C01838=1166.104,19.799,-47.480,-179.912,6.031,149.056
C01839=1166.100,20.048,-47.495,-179.910,6.031,149.055
C01840=1166.094,20.297,-47.509,-179.907,6.032,149.055
C01841=1166.089,20.547,-47.523,-179.905,6.033,149.054
C01842=1166.084,20.797,-47.538,-179.902,6.033,149.053
C01843=1166.078,21.047,-47.553,-179.899,6.034,149.053
C01844=1166.073,21.297,-47.567,-179.897,6.035,149.052
C01845=1166.069,21.546,-47.582,-179.894,6.036,149.052
C01846=1166.063,21.795,-47.596,-179.892,6.037,149.051
C01847=1166.058,22.044,-47.610,-179.889,6.037,149.051
C01848=1166.053,22.294,-47.624,-179.887,6.038,149.050
C01849=1166.048,22.544,-47.639,-179.884,6.039,149.049
C01850=1166.044,22.793,-47.654,-179.881,6.040,149.049
C01851=1166.038,23.043,-47.668,-179.879,6.041,149.048
C01852=1166.033,23.293,-47.683,-179.877,6.041,149.048
C01853=1166.028,23.542,-47.697,-179.874,6.042,149.047
C01854=1166.023,23.791,-47.712,-179.871,6.043,149.046
C01855=1166.018,24.040,-47.726,-179.869,6.044,149.046
C01856=1166.013,24.290,-47.740,-179.866,6.044,149.045
C01857=1166.008,24.540,-47.754,-179.864,6.045,149.045
C01858=1166.003,24.789,-47.770,-179.862,6.046,149.044
C01859=1165.998,25.039,-47.784,-179.858,6.047,149.043
C01860=1165.993,25.289,-47.799,-179.856,6.048,149.043
C01861=1165.988,25.538,-47.814,-179.853,6.048,149.042
C01862=1165.983,25.787,-47.828,-179.851,6.049,149.042
C01863=1165.977,26.037,-47.843,-179.849,6.050,149.041
C01864=1165.973,26.287,-47.858,-179.846,6.051,149.041
C01865=1165.968,26.536,-47.872,-179.843,6.052,149.040
C01866=1165.963,26.786,-47.886,-179.841,6.052,149.039
C01867=1165.957,27.035,-47.901,-179.838,6.053,149.039
C01868=1165.952,27.284,-47.916,-179.835,6.054,149.038
C01869=1165.947,27.534,-47.930,-179.833,6.055,149.038
C01870=1165.942,27.803,-47.946,-179.830,6.056,149.037
C01871=1165.936,28.072,-47.962,-179.827,6.057,149.036
C01872=1165.931,28.341,-47.978,-179.825,6.058,149.036
C01873=1165.925,28.610,-47.994,-179.822,6.058,149.035
C01874=1165.920,28.859,-48.009,-179.819,6.060,149.035
C01875=1165.915,29.109,-48.023,-179.817,6.060,149.034
C01876=1165.911,29.358,-48.038,-179.814,6.061,149.034
C01877=1165.905,29.608,-48.053,-179.812,6.062,149.033
C01878=1165.900,29.857,-48.068,-179.809,6.062,149.032
C01879=1165.895,30.107,-48.082,-179.807,6.064,149.032
C01880=1165.890,30.357,-48.097,-179.804,6.064,149.031
C01881=1165.885,30.606,-48.112,-179.801,6.065,149.031
C01882=1165.880,30.855,-48.127,-179.799,6.066,149.030
C01883=1165.875,31.105,-48.142,-179.796,6.067,149.029
C01884=1165.870,31.354,-48.157,-179.794,6.068,149.029
C01885=1165.865,31.604,-48.171,-179.791,6.068,149.028
C01886=1165.860,31.853,-48.187,-179.789,6.069,149.028
C01887=1165.855,32.103,-48.201,-179.786,6.070,149.027
C01888=1165.850,32.352,-48.216,-179.784,6.071,149.027
C01889=1165.844,32.602,-48.231,-179.781,6.072,149.026
C01890=1165.840,32.851,-48.246,-179.779,6.073,149.026
C01891=1165.834,33.101,-48.261,-179.776,6.074,149.025
C01892=1165.829,33.350,-48.276,-179.773,6.074,149.024
C01893=1165.825,33.599,-48.291,-179.771,6.075,149.024
C01894=1165.820,33.850,-48.306,-179.768,6.076,149.023
C01895=1165.815,34.099,-48.321,-179.765,6.077,149.023
C01896=1165.810,34.348,-48.337,-179.763,6.078,149.022
C01897=1165.805,34.598,-48.351,-179.761,6.079,149.022
C01898=1165.799,34.847,-48.367,-179.758,6.079,149.021
C01899=1165.794,35.097,-48.381,-179.755,6.081,149.020
C01900=1165.790,35.346,-48.396,-179.753,6.081,149.020
C01901=1165.784,35.596,-48.412,-179.750,6.082,149.019
C01902=1165.780,35.845,-48.427,-179.747,6.084,149.019
C01903=1165.774,36.095,-48.441,-179.745,6.084,149.018
C01904=1165.769,36.344,-48.456,-179.742,6.085,149.018
C01905=1165.764,36.593,-48.472,-179.740,6.085,149.017
C01906=1165.760,36.844,-48.487,-179.737,6.087,149.016
C01907=1165.754,37.093,-48.502,-179.734,6.087,149.016
C01908=1165.750,37.342,-48.517,-179.732,6.088,149.015
C01909=1165.744,37.592,-48.533,-179.730,6.089,149.015
C01910=1165.739,37.841,-48.547,-179.727,6.090,149.014
C01911=1165.734,38.091,-48.563,-179.724,6.091,149.014
C01912=1165.729,38.340,-48.578,-179.722,6.092,149.013
C01913=1165.724,38.589,-48.593,-179.719,6.093,149.012
C01914=1165.719,38.840,-48.608,-179.717,6.094,149.012
C01915=1165.714,39.089,-48.623,-179.714,6.094,149.011
C01916=1165.709,39.338,-48.639,-179.711,6.096,149.011
C01917=1165.704,39.587,-48.654,-179.709,6.097,149.010
C01918=1165.699,39.837,-48.670,-179.706,6.097,149.010
C01919=1165.694,40.086,-48.685,-179.704,6.098,149.009
C01920=1165.688,40.336,-48.700,-179.701,6.100,149.009
C01921=1165.684,40.586,-48.715,-179.698,6.100,149.008
C01922=1165.679,40.835,-48.730,-179.696,6.101,149.007
C01923=1165.673,41.085,-48.746,-179.693,6.102,149.007
C01924=1165.669,41.334,-48.761,-179.690,6.103,149.006
C01925=1165.663,41.583,-48.777,-179.688,6.104,149.006
C01926=1165.659,41.833,-48.792,-179.685,6.105,149.005
C01927=1165.654,42.082,-48.808,-179.683,6.106,149.005
C01928=1165.649,42.332,-48.823,-179.680,6.106,149.004
C01929=1165.644,42.581,-48.837,-179.678,6.107,149.003
C01930=1165.638,42.831,-48.853,-179.675,6.108,149.003
C01931=1165.633,43.081,-48.869,-179.673,6.109,149.002
C01932=1165.629,43.330,-48.884,-179.670,6.110,149.002
C01933=1165.623,43.579,-48.900,-179.667,6.111,149.001
C01934=1165.618,43.829,-48.915,-179.665,6.112,149.001
C01935=1165.613,44.078,-48.930,-179.662,6.113,149.000
C01936=1165.609,44.328,-48.946,-179.659,6.114,148.999
C01937=1165.603,44.577,-48.962,-179.657,6.115,148.999
C01938=1165.599,44.827,-48.977,-179.654,6.115,148.998
C01939=1165.593,45.076,-48.992,-179.652,6.117,148.998
C01940=1165.588,45.326,-49.008,-179.649,6.118,148.997
C01941=1165.584,45.575,-49.023,-179.647,6.118,148.997
C01942=1165.578,45.825,-49.039,-179.644,6.120,148.996
C01943=1165.573,46.074,-49.054,-179.641,6.121,148.996
C01944=1165.568,46.323,-49.071,-179.639,6.121,148.995
C01945=1165.564,46.572,-49.086,-179.636,6.123,148.995
C01946=1165.558,46.822,-49.102,-179.633,6.123,148.994
C01947=1165.554,47.072,-49.118,-179.631,6.124,148.993
C01948=1165.548,47.321,-49.133,-179.628,6.125,148.993
C01949=1165.544,47.570,-49.148,-179.626,6.126,148.992
C01950=1165.538,47.820,-49.164,-179.623,6.127,148.992
C01951=1165.533,48.070,-49.180,-179.621,6.128,148.991
C01952=1165.528,48.319,-49.195,-179.618,6.129,148.991
C01953=1165.524,48.568,-49.211,-179.616,6.130,148.990
C01954=1165.519,48.818,-49.227,-179.613,6.131,148.989
C01955=1165.514,49.067,-49.243,-179.610,6.132,148.989
C01956=1165.508,49.317,-49.258,-179.608,6.132,148.988
C01957=1165.503,49.567,-49.274,-179.605,6.134,148.988
C01958=1165.499,49.816,-49.289,-179.602,6.135,148.987
C01959=1165.494,50.065,-49.305,-179.600,6.136,148.987
C01960=1165.489,50.315,-49.321,-179.597,6.137,148.986
C01961=1165.483,50.564,-49.337,-179.595,6.138,148.986
C01962=1165.478,50.814,-49.353,-179.592,6.139,148.985
C01963=1165.474,51.063,-49.369,-179.589,6.140,148.985
C01964=1165.469,51.312,-49.384,-179.587,6.140,148.984
C01965=1165.464,51.562,-49.400,-179.584,6.142,148.983
C01966=1165.459,51.812,-49.416,-179.581,6.142,148.983
C01967=1165.454,52.061,-49.432,-179.579,6.143,148.982
C01968=1165.449,52.311,-49.448,-179.576,6.145,148.982
C01969=1165.444,52.560,-49.464,-179.574,6.145,148.981
C01970=1165.438,52.809,-49.480,-179.571,6.147,148.981
C01971=1165.434,53.059,-49.496,-179.568,6.148,148.980
C01972=1165.428,53.308,-49.511,-179.566,6.148,148.979
C01973=1165.424,53.557,-49.527,-179.563,6.150,148.979
C01974=1165.419,53.826,-49.545,-179.560,6.150,148.978
C01975=1165.413,54.094,-49.562,-179.557,6.152,148.978
C01976=1165.408,54.363,-49.579,-179.555,6.152,148.977
C01977=1165.402,54.631,-49.596,-179.552,6.154,148.977
C01978=1165.398,54.882,-49.612,-179.549,6.154,148.976
C01979=1165.392,55.130,-49.628,-179.546,6.156,148.975
C01980=1165.388,55.380,-49.644,-179.544,6.156,148.975
C01981=1165.383,55.629,-49.660,-179.541,6.158,148.974
C01982=1165.378,55.879,-49.676,-179.539,6.159,148.974
C01983=1165.373,56.128,-49.692,-179.536,6.159,148.973
C01984=1165.367,56.377,-49.708,-179.534,6.161,148.973
C01985=1165.363,56.628,-49.724,-179.531,6.162,148.972
C01986=1165.357,56.876,-49.740,-179.528,6.163,148.972
C01987=1165.353,57.126,-49.756,-179.526,6.164,148.971
C01988=1165.348,57.375,-49.772,-179.523,6.165,148.971
C01989=1165.343,57.625,-49.788,-179.520,6.166,148.970
C01990=1165.338,57.874,-49.805,-179.518,6.167,148.969
C01991=1165.333,58.124,-49.821,-179.515,6.168,148.969
C01992=1165.328,58.373,-49.837,-179.513,6.169,148.968
C01993=1165.322,58.623,-49.854,-179.510,6.170,148.968
C01994=1165.317,58.872,-49.870,-179.507,6.171,148.967
C01995=1165.312,59.122,-49.886,-179.505,6.172,148.967
C01996=1165.307,59.371,-49.902,-179.502,6.173,148.966
C01997=1165.303,59.621,-49.919,-179.499,6.174,148.966
C01998=1165.298,59.870,-49.934,-179.497,6.176,148.965
C01999=1165.293,60.119,-49.951,-179.494,6.176,148.964
C02000=1165.288,60.369,-49.967,-179.492,6.177,148.964
C02001=1165.283,60.618,-49.983,-179.489,6.179,148.964
C02002=1165.278,60.867,-50.000,-179.486,6.179,148.963
C02003=1165.273,61.117,-50.016,-179.484,6.181,148.962
C02004=1165.268,61.366,-50.032,-179.481,6.181,148.962
C02005=1165.263,61.616,-50.048,-179.478,6.183,148.961
C02006=1165.258,61.865,-50.065,-179.476,6.183,148.961
C02007=1165.253,62.115,-50.081,-179.473,6.184,148.960
C02008=1165.248,62.364,-50.097,-179.470,6.186,148.960
C02009=1165.243,62.614,-50.114,-179.468,6.187,148.959
C02010=1165.238,62.862,-50.130,-179.465,6.188,148.958
C02011=1165.233,63.112,-50.147,-179.463,6.189,148.958
C02012=1165.228,63.362,-50.163,-179.460,6.190,148.958
C02013=1165.223,63.611,-50.179,-179.457,6.191,148.957
C02014=1165.219,63.861,-50.196,-179.455,6.193,148.957
C02015=1165.213,64.110,-50.212,-179.452,6.193,148.956
C02016=1165.209,64.359,-50.228,-179.450,6.194,148.955
C02017=1165.203,64.609,-50.245,-179.447,6.195,148.955
C02018=1165.198,64.858,-50.262,-179.444,6.196,148.954
C02019=1165.194,65.108,-50.278,-179.441,6.197,148.954
C02020=1165.189,65.357,-50.294,-179.439,6.198,148.953
C02021=1165.183,65.607,-50.311,-179.436,6.200,148.953
C02022=1165.178,65.855,-50.328,-179.434,6.200,148.952
C02023=1165.174,66.105,-50.344,-179.431,6.202,148.952
C02024=1165.169,66.354,-50.361,-179.428,6.203,148.951
C02025=1165.163,66.604,-50.377,-179.426,6.204,148.951
C02026=1165.159,66.854,-50.394,-179.423,6.205,148.950
C02027=1165.154,67.103,-50.411,-179.420,6.207,148.950
C02028=1165.149,67.352,-50.427,-179.418,6.207,148.949
C02029=1165.144,67.602,-50.444,-179.415,6.209,148.948
C02030=1165.139,67.850,-50.460,-179.412,6.209,148.948
C02031=1165.134,68.100,-50.477,-179.410,6.210,148.947
C02032=1165.130,68.350,-50.493,-179.407,6.212,148.947
C02033=1165.124,68.599,-50.510,-179.405,6.212,148.946
C02034=1165.119,68.849,-50.527,-179.402,6.214,148.946
C02035=1165.115,69.098,-50.543,-179.399,6.215,148.945
C02036=1165.109,69.347,-50.560,-179.397,6.216,148.945
C02037=1165.105,69.597,-50.577,-179.394,6.217,148.944
C02038=1165.100,69.846,-50.594,-179.391,6.218,148.944
C02039=1165.094,70.095,-50.610,-179.389,6.219,148.943
C02040=1165.090,70.345,-50.627,-179.386,6.221,148.943
C02041=1165.085,70.595,-50.644,-179.384,6.221,148.942
C02042=1165.080,70.844,-50.661,-179.381,6.223,148.941
C02043=1165.075,71.093,-50.677,-179.378,6.224,148.941
C02044=1165.070,71.343,-50.695,-179.375,6.225,148.940
C02045=1165.065,71.592,-50.711,-179.373,6.226,148.940
C02046=1165.060,71.841,-50.728,-179.370,6.228,148.939
C02047=1165.055,72.091,-50.745,-179.368,6.228,148.939
C02048=1165.050,72.340,-50.762,-179.365,6.230,148.938
C02049=1165.045,72.589,-50.778,-179.362,6.230,148.938
C02050=1165.040,72.839,-50.795,-179.360,6.232,148.937
C02051=1165.035,73.089,-50.812,-179.357,6.232,148.937
C02052=1165.031,73.337,-50.830,-179.354,6.234,148.936
C02053=1165.026,73.586,-50.846,-179.352,6.235,148.936
C02054=1165.021,73.836,-50.863,-179.349,6.236,148.935
C02055=1165.016,74.085,-50.880,-179.347,6.237,148.935
C02056=1165.011,74.335,-50.897,-179.343,6.239,148.934
C02057=1165.006,74.584,-50.914,-179.341,6.239,148.934
C02058=1165.001,74.834,-50.931,-179.339,6.241,148.933
C02059=1164.996,75.083,-50.947,-179.336,6.242,148.933
C02060=1164.991,75.333,-50.965,-179.333,6.243,148.932
C02061=1164.987,75.582,-50.982,-179.330,6.245,148.931
C02062=1164.981,75.831,-50.999,-179.328,6.246,148.931
C02063=1164.976,76.081,-51.016,-179.325,6.247,148.931
C02064=1164.971,76.330,-51.033,-179.322,6.248,148.930
C02065=1164.967,76.579,-51.050,-179.320,6.249,148.930
C02066=1164.962,76.829,-51.068,-179.317,6.250,148.929
C02067=1164.957,77.078,-51.084,-179.314,6.252,148.928
C02068=1164.951,77.328,-51.101,-179.312,6.252,148.928
C02069=1164.947,77.577,-51.119,-179.309,6.254,148.927
C02070=1164.942,77.826,-51.136,-179.307,6.255,148.927
C02071=1164.937,78.076,-51.153,-179.304,6.256,148.926
C02072=1164.932,78.324,-51.170,-179.302,6.257,148.926
C02073=1164.927,78.574,-51.187,-179.299,6.259,148.925
C02074=1164.922,78.823,-51.204,-179.296,6.260,148.925
C02075=1164.917,79.073,-51.221,-179.293,6.261,148.924
C02076=1164.912,79.322,-51.239,-179.290,6.262,148.924
C02077=1164.908,79.572,-51.256,-179.288,6.263,148.923
C02078=1164.902,79.840,-51.274,-179.285,6.264,148.923
C02079=1164.897,80.108,-51.294,-179.282,6.266,148.922
C02080=1164.892,80.377,-51.312,-179.280,6.267,148.922
C02081=1164.886,80.645,-51.330,-179.277,6.268,148.921
C02082=1164.881,80.895,-51.347,-179.274,6.270,148.920
C02083=1164.877,81.144,-51.365,-179.271,6.270,148.920
C02084=1164.871,81.394,-51.382,-179.269,6.272,148.920
C02085=1164.867,81.643,-51.400,-179.266,6.273,148.919
C02086=1164.862,81.892,-51.417,-179.263,6.274,148.919
C02087=1164.857,82.141,-51.435,-179.260,6.276,148.918
C02088=1164.851,82.390,-51.452,-179.258,6.277,148.917
C02089=1164.847,82.640,-51.468,-179.255,6.278,148.917
C02090=1164.842,82.889,-51.486,-179.253,6.279,148.916
C02091=1164.837,83.139,-51.503,-179.250,6.280,148.916
C02092=1164.832,83.388,-51.521,-179.247,6.281,148.915
C02093=1164.827,83.638,-51.538,-179.245,6.283,148.915
C02094=1164.822,83.887,-51.556,-179.242,6.284,148.914
C02095=1164.817,84.137,-51.573,-179.239,6.285,148.914
C02096=1164.812,84.386,-51.591,-179.236,6.287,148.913
C02097=1164.808,84.635,-51.609,-179.234,6.287,148.913
C02098=1164.803,84.884,-51.626,-179.231,6.289,148.912
C02099=1164.798,85.134,-51.644,-179.228,6.290,148.912
C02100=1164.793,85.383,-51.661,-179.226,6.291,148.911
C02101=1164.789,85.632,-51.679,-179.223,6.293,148.911
C02102=1164.783,85.882,-51.696,-179.221,6.294,148.910
C02103=1164.778,86.131,-51.714,-179.218,6.295,148.910
C02104=1164.773,86.380,-51.731,-179.215,6.297,148.909
C02105=1164.768,86.629,-51.749,-179.213,6.298,148.909
C02106=1164.764,86.878,-51.766,-179.210,6.299,148.908
C02107=1164.758,87.128,-51.783,-179.207,6.300,148.908
C02108=1164.753,87.377,-51.801,-179.205,6.301,148.907
C02109=1164.748,87.626,-51.819,-179.201,6.303,148.907
C02110=1164.743,87.876,-51.837,-179.199,6.304,148.906
C02111=1164.738,88.125,-51.855,-179.197,6.305,148.906
C02112=1164.734,88.374,-51.872,-179.194,6.306,148.905
C02113=1164.729,88.624,-51.890,-179.191,6.308,148.905
C02114=1164.724,88.873,-51.907,-179.188,6.309,148.904
C02115=1164.719,89.122,-51.925,-179.186,6.310,148.904
C02116=1164.714,89.372,-51.943,-179.183,6.311,148.903
C02117=1164.710,89.622,-51.961,-179.180,6.313,148.903
C02118=1164.705,89.871,-51.979,-179.178,6.314,148.902
C02119=1164.700,90.121,-51.997,-179.175,6.315,148.902
C02120=1164.696,90.369,-52.014,-179.173,6.316,148.901
C02121=1164.691,90.619,-52.032,-179.170,6.318,148.901
C02122=1164.685,90.868,-52.049,-179.167,6.319,148.900
C02123=1164.681,91.118,-52.067,-179.164,6.320,148.900
C02124=1164.676,91.367,-52.085,-179.162,6.322,148.899
C02125=1164.671,91.616,-52.103,-179.159,6.323,148.899
C02126=1164.666,91.865,-52.121,-179.156,6.324,148.898
C02127=1164.661,92.115,-52.139,-179.154,6.325,148.898
C02128=1164.656,92.364,-52.157,-179.151,6.326,148.897
C02129=1164.651,92.613,-52.175,-179.148,6.328,148.897
C02130=1164.646,92.862,-52.193,-179.146,6.329,148.896
C02131=1164.641,93.112,-52.211,-179.143,6.330,148.896
C02132=1164.637,93.361,-52.229,-179.140,6.332,148.895
C02133=1164.632,93.611,-52.247,-179.137,6.333,148.895
C02134=1164.627,93.860,-52.265,-179.135,6.334,148.894
C02135=1164.622,94.109,-52.283,-179.132,6.336,148.894
C02136=1164.617,94.359,-52.300,-179.129,6.337,148.893
C02137=1164.612,94.608,-52.318,-179.127,6.338,148.893
C02138=1164.607,94.857,-52.336,-179.124,6.340,148.892
C02139=1164.602,95.106,-52.354,-179.121,6.341,148.892
C02140=1164.597,95.355,-52.372,-179.119,6.342,148.891
C02141=1164.593,95.605,-52.390,-179.116,6.343,148.891
C02142=1164.588,95.855,-52.408,-179.113,6.345,148.890
C02143=1164.583,96.104,-52.426,-179.111,6.346,148.890
C02144=1164.578,96.353,-52.444,-179.108,6.348,148.890
C02145=1164.573,96.602,-52.462,-179.105,6.349,148.889
C02146=1164.567,96.852,-52.481,-179.103,6.350,148.889
C02147=1164.563,97.101,-52.499,-179.100,6.352,148.888
C02148=1164.558,97.351,-52.517,-179.097,6.353,148.887
C02149=1164.553,97.600,-52.535,-179.095,6.354,148.887
C02150=1164.549,97.848,-52.554,-179.092,6.356,148.887
C02151=1164.544,98.097,-52.572,-179.089,6.357,148.886
C02152=1164.539,98.347,-52.590,-179.087,6.358,148.886
C02153=1164.535,98.597,-52.608,-179.084,6.360,148.885
C02154=1164.530,98.846,-52.626,-179.081,6.361,148.885
C02155=1164.524,99.095,-52.645,-179.079,6.362,148.884
C02156=1164.519,99.344,-52.663,-179.076,6.363,148.884
C02157=1164.514,99.594,-52.681,-179.073,6.365,148.883
C02158=1164.510,99.843,-52.700,-179.071,6.366,148.883
C02159=1164.505,100.092,-52.718,-179.068,6.367,148.882
C02160=1164.500,100.341,-52.736,-179.065,6.369,148.882
C02161=1164.495,100.591,-52.754,-179.062,6.370,148.881
C02162=1164.490,100.841,-52.773,-179.060,6.371,148.881
C02163=1164.485,101.090,-52.791,-179.057,6.373,148.880
C02164=1164.481,101.338,-52.809,-179.055,6.375,148.880
C02165=1164.475,101.588,-52.828,-179.052,6.375,148.879
C02166=1164.470,101.837,-52.846,-179.049,6.377,148.879
C02167=1164.466,102.087,-52.864,-179.047,6.379,148.878
C02168=1164.461,102.335,-52.883,-179.044,6.379,148.878
C02169=1164.456,102.585,-52.901,-179.041,6.381,148.877
C02170=1164.451,102.835,-52.920,-179.038,6.383,148.877
C02171=1164.447,103.084,-52.938,-179.036,6.384,148.877
C02172=1164.442,103.332,-52.956,-179.033,6.385,148.876
C02173=1164.436,103.582,-52.975,-179.030,6.387,148.876
C02174=1164.432,103.832,-52.993,-179.028,6.388,148.875
C02175=1164.427,104.080,-53.012,-179.025,6.389,148.874
C02176=1164.422,104.330,-53.030,-179.022,6.391,148.874
C02177=1164.417,104.580,-53.049,-179.020,6.392,148.874
C02178=1164.413,104.828,-53.068,-179.017,6.394,148.873
C02179=1164.408,105.077,-53.086,-179.014,6.395,148.873
C02180=1164.403,105.326,-53.105,-179.012,6.396,148.872
C02181=1164.398,105.576,-53.123,-179.009,6.398,148.872
C02182=1164.392,105.845,-53.143,-179.006,6.399,148.871
C02183=1164.388,106.112,-53.163,-179.003,6.401,148.871
C02184=1164.382,106.382,-53.184,-179.000,6.402,148.870
C02185=1164.377,106.650,-53.203,-178.997,6.404,148.870
C02186=1164.372,106.899,-53.223,-178.995,6.405,148.869
C02187=1164.368,107.149,-53.241,-178.992,6.407,148.869
C02188=1164.363,107.397,-53.260,-178.989,6.408,148.868
C02189=1164.357,107.647,-53.278,-178.986,6.410,148.868
C02190=1164.353,107.896,-53.297,-178.984,6.411,148.867
C02191=1164.348,108.145,-53.316,-178.981,6.412,148.867
C02192=1164.343,108.394,-53.334,-178.978,6.414,148.866
C02193=1164.339,108.644,-53.353,-178.975,6.415,148.866
C02194=1164.333,108.893,-53.372,-178.973,6.416,148.866
C02195=1164.329,109.142,-53.390,-178.970,6.418,148.865
C02196=1164.324,109.391,-53.410,-178.967,6.419,148.865
C02197=1164.319,109.641,-53.428,-178.965,6.421,148.864
C02198=1164.314,109.890,-53.447,-178.963,6.422,148.864
C02199=1164.309,110.139,-53.465,-178.960,6.424,148.863
C02200=1164.304,110.388,-53.485,-178.957,6.425,148.863
C02201=1164.300,110.638,-53.504,-178.954,6.427,148.862
C02202=1164.295,110.887,-53.522,-178.952,6.428,148.862
C02203=1164.290,111.136,-53.541,-178.949,6.429,148.861
C02204=1164.285,111.385,-53.559,-178.946,6.431,148.861
C02205=1164.281,111.635,-53.579,-178.943,6.432,148.860
C02206=1164.275,111.884,-53.598,-178.940,6.434,148.860
C02207=1164.270,112.133,-53.616,-178.938,6.435,148.860
C02208=1164.266,112.383,-53.636,-178.935,6.436,148.859
C02209=1164.261,112.631,-53.655,-178.932,6.438,148.859
C02210=1164.256,112.881,-53.674,-178.930,6.440,148.858
C02211=1164.251,113.130,-53.692,-178.928,6.441,148.858
C02212=1164.247,113.380,-53.712,-178.924,6.442,148.857
C02213=1164.242,113.628,-53.731,-178.922,6.444,148.857
C02214=1164.237,113.878,-53.750,-178.919,6.446,148.856
C02215=1164.232,114.127,-53.769,-178.916,6.447,148.856
C02216=1164.228,114.376,-53.788,-178.914,6.448,148.855
C02217=1164.222,114.625,-53.807,-178.911,6.450,148.855
C02218=1164.218,114.875,-53.826,-178.908,6.451,148.854
C02219=1164.213,115.124,-53.845,-178.905,6.453,148.854
C02220=1164.208,115.374,-53.864,-178.903,6.455,148.854
C02221=1164.203,115.622,-53.883,-178.901,6.456,148.853
C02222=1164.199,115.872,-53.903,-178.897,6.457,148.853
C02223=1164.193,116.121,-53.922,-178.895,6.459,148.852
C02224=1164.189,116.370,-53.940,-178.892,6.460,148.852
C02225=1164.184,116.619,-53.960,-178.889,6.462,148.851
C02226=1164.179,116.869,-53.979,-178.887,6.463,148.851
C02227=1164.174,117.117,-53.998,-178.884,6.464,148.850
C02228=1164.169,117.367,-54.018,-178.881,6.466,148.850
C02229=1164.164,117.616,-54.037,-178.879,6.468,148.850
C02230=1164.160,117.865,-54.056,-178.876,6.470,148.849
C02231=1164.155,118.114,-54.075,-178.873,6.471,148.849
C02232=1164.150,118.364,-54.094,-178.870,6.472,148.848
C02233=1164.145,118.613,-54.113,-178.868,6.473,148.848
C02234=1164.140,118.862,-54.133,-178.865,6.475,148.847
C02235=1164.136,119.112,-54.152,-178.862,6.477,148.847
C02236=1164.130,119.361,-54.172,-178.860,6.479,148.847
C02237=1164.126,119.610,-54.191,-178.857,6.479,148.846
C02238=1164.121,119.859,-54.210,-178.854,6.481,148.845
C02239=1164.116,120.108,-54.230,-178.852,6.483,148.845
C02240=1164.111,120.358,-54.249,-178.849,6.484,148.845
C02241=1164.107,120.607,-54.268,-178.846,6.486,148.844
C02242=1164.102,120.856,-54.288,-178.843,6.487,148.844
C02243=1164.097,121.105,-54.307,-178.840,6.489,148.843
C02244=1164.092,121.355,-54.327,-178.838,6.490,148.843
C02245=1164.088,121.603,-54.346,-178.835,6.492,148.842
C02246=1164.083,121.852,-54.366,-178.833,6.494,148.842
C02247=1164.078,122.102,-54.385,-178.830,6.495,148.842
C02248=1164.073,122.350,-54.405,-178.827,6.497,148.841
C02249=1164.068,122.600,-54.424,-178.824,6.498,148.841
C02250=1164.063,122.850,-54.444,-178.822,6.499,148.840
C02251=1164.059,123.098,-54.463,-178.819,6.501,148.840
C02252=1164.054,123.348,-54.482,-178.817,6.503,148.839
C02253=1164.049,123.597,-54.502,-178.814,6.504,148.839
C02254=1164.044,123.846,-54.522,-178.811,6.506,148.838
C02255=1164.039,124.095,-54.542,-178.808,6.507,148.838
C02256=1164.035,124.345,-54.561,-178.805,6.509,148.838
C02257=1164.029,124.594,-54.581,-178.803,6.510,148.837
C02258=1164.025,124.843,-54.600,-178.800,6.512,148.837
C02259=1164.021,125.092,-54.620,-178.798,6.514,148.836
C02260=1164.016,125.341,-54.639,-178.794,6.515,148.836
C02261=1164.011,125.590,-54.659,-178.792,6.517,148.835
C02262=1164.006,125.840,-54.679,-178.789,6.518,148.835
C02263=1164.002,126.089,-54.699,-178.786,6.520,148.835
C02264=1163.996,126.338,-54.718,-178.784,6.522,148.834
C02265=1163.992,126.587,-54.738,-178.781,6.523,148.834
C02266=1163.987,126.837,-54.758,-178.779,6.524,148.833
C02267=1163.982,127.085,-54.778,-178.776,6.526,148.833
C02268=1163.977,127.335,-54.797,-178.773,6.528,148.832
C02269=1163.972,127.584,-54.817,-178.770,6.529,148.832
C02270=1163.968,127.833,-54.837,-178.767,6.531,148.832
C02271=1163.963,128.082,-54.857,-178.765,6.533,148.831
C02272=1163.958,128.331,-54.876,-178.762,6.534,148.831
C02273=1163.953,128.580,-54.897,-178.759,6.536,148.830
C02274=1163.949,128.830,-54.916,-178.757,6.537,148.830
C02275=1163.944,129.078,-54.936,-178.754,6.538,148.829
C02276=1163.939,129.328,-54.956,-178.751,6.540,148.829
C02277=1163.934,129.577,-54.976,-178.749,6.542,148.829
C02278=1163.930,129.826,-54.996,-178.746,6.544,148.828
C02279=1163.925,130.076,-55.016,-178.743,6.545,148.828
C02280=1163.920,130.324,-55.036,-178.740,6.547,148.827
C02281=1163.915,130.574,-55.055,-178.738,6.549,148.827
C02282=1163.911,130.823,-55.076,-178.735,6.550,148.826
C02283=1163.906,131.072,-55.095,-178.732,6.552,148.826
C02284=1163.901,131.320,-55.115,-178.729,6.554,148.826
C02285=1163.896,131.570,-55.135,-178.727,6.555,148.825
C02286=1163.891,131.839,-55.157,-178.724,6.557,148.825
C02287=1163.886,132.107,-55.178,-178.721,6.559,148.824
C02288=1163.880,132.376,-55.200,-178.718,6.560,148.824
C02289=1163.875,132.645,-55.221,-178.715,6.562,148.823
C02290=1163.871,132.894,-55.242,-178.712,6.564,148.823
C02291=1163.866,133.143,-55.262,-178.710,6.565,148.823
C02292=1163.861,133.392,-55.282,-178.707,6.567,148.822
C02293=1163.857,133.641,-55.303,-178.704,6.569,148.822
C02294=1163.851,133.890,-55.322,-178.701,6.570,148.821
C02295=1163.847,134.139,-55.342,-178.698,6.572,148.821
C02296=1163.842,134.389,-55.362,-178.696,6.574,148.820
C02297=1163.838,134.638,-55.382,-178.694,6.575,148.820
C02298=1163.832,134.887,-55.403,-178.691,6.576,148.820
C02299=1163.828,135.137,-55.423,-178.688,6.578,148.819
C02300=1163.823,135.385,-55.443,-178.685,6.580,148.819
C02301=1163.819,135.634,-55.464,-178.683,6.581,148.818
C02302=1163.813,135.883,-55.483,-178.680,6.583,148.818
C02303=1163.808,136.133,-55.504,-178.677,6.585,148.818
C02304=1163.804,136.382,-55.524,-178.675,6.587,148.817
C02305=1163.799,136.630,-55.545,-178.671,6.588,148.817
C02306=1163.795,136.880,-55.564,-178.669,6.590,148.816
C02307=1163.789,137.129,-55.585,-178.666,6.591,148.816
C02308=1163.785,137.378,-55.606,-178.663,6.593,148.816
C02309=1163.781,137.627,-55.626,-178.661,6.595,148.815
C02310=1163.776,137.877,-55.646,-178.658,6.597,148.815
C02311=1163.771,138.126,-55.667,-178.655,6.598,148.814
C02312=1163.766,138.375,-55.687,-178.653,6.600,148.814
C02313=1163.761,138.623,-55.707,-178.650,6.602,148.814
C02314=1163.756,138.872,-55.728,-178.647,6.604,148.813
C02315=1163.751,139.122,-55.748,-178.644,6.605,148.813
C02316=1163.747,139.371,-55.768,-178.642,6.607,148.812
C02317=1163.742,139.620,-55.789,-178.639,6.609,148.812
C02318=1163.737,139.869,-55.809,-178.636,6.611,148.812
C02319=1163.733,140.118,-55.830,-178.633,6.612,148.811
C02320=1163.728,140.367,-55.851,-178.630,6.614,148.811
C02321=1163.723,140.616,-55.871,-178.628,6.615,148.810
C02322=1163.718,140.866,-55.891,-178.625,6.617,148.810
C02323=1163.713,141.115,-55.912,-178.623,6.618,148.809
C02324=1163.709,141.364,-55.932,-178.620,6.620,148.809
C02325=1163.704,141.613,-55.952,-178.617,6.622,148.809
C02326=1163.699,141.862,-55.973,-178.615,6.623,148.808
C02327=1163.695,142.111,-55.994,-178.612,6.625,148.808
C02328=1163.690,142.361,-56.015,-178.609,6.627,148.808
C02329=1163.685,142.609,-56.035,-178.607,6.628,148.807
C02330=1163.680,142.859,-56.056,-178.604,6.630,148.807
C02331=1163.676,143.108,-56.076,-178.601,6.632,148.806
C02332=1163.671,143.357,-56.097,-178.599,6.634,148.806
C02333=1163.666,143.606,-56.118,-178.596,6.635,148.806
C02334=1163.662,143.855,-56.138,-178.593,6.637,148.805
C02335=1163.657,144.105,-56.159,-178.590,6.639,148.805
C02336=1163.653,144.354,-56.180,-178.588,6.641,148.804
C02337=1163.647,144.603,-56.201,-178.585,6.642,148.804
C02338=1163.643,144.852,-56.221,-178.582,6.644,148.804
C02339=1163.638,145.101,-56.243,-178.580,6.646,148.803
C02340=1163.634,145.350,-56.263,-178.577,6.648,148.803
C02341=1163.628,145.599,-56.284,-178.574,6.650,148.803
C02342=1163.624,145.848,-56.305,-178.571,6.652,148.802
C02343=1163.619,146.097,-56.325,-178.568,6.654,148.802
C02344=1163.614,146.346,-56.346,-178.566,6.655,148.801
C02345=1163.609,146.595,-56.367,-178.563,6.657,148.801
C02346=1163.605,146.844,-56.388,-178.560,6.658,148.800
C02347=1163.600,147.093,-56.409,-178.557,6.660,148.800
C02348=1163.596,147.342,-56.430,-178.554,6.662,148.800
C02349=1163.591,147.592,-56.451,-178.552,6.664,148.799
C02350=1163.586,147.841,-56.472,-178.549,6.665,148.799
C02351=1163.582,148.089,-56.493,-178.546,6.667,148.799
C02352=1163.576,148.339,-56.514,-178.543,6.669,148.798
C02353=1163.572,148.588,-56.534,-178.541,6.671,148.798
C02354=1163.567,148.837,-56.555,-178.538,6.672,148.797
C02355=1163.562,149.085,-56.577,-178.535,6.674,148.797
C02356=1163.558,149.335,-56.597,-178.533,6.676,148.797
C02357=1163.553,149.584,-56.618,-178.530,6.678,148.796
C02358=1163.548,149.834,-56.639,-178.527,6.679,148.796
C02359=1163.544,150.082,-56.660,-178.525,6.681,148.795
C02360=1163.538,150.331,-56.681,-178.522,6.683,148.795
C02361=1163.533,150.580,-56.702,-178.519,6.684,148.795
C02362=1163.530,150.829,-56.724,-178.517,6.687,148.795
C02363=1163.525,151.079,-56.745,-178.514,6.688,148.794
C02364=1163.519,151.328,-56.766,-178.512,6.690,148.794
C02365=1163.515,151.576,-56.787,-178.509,6.692,148.793
C02366=1163.510,151.826,-56.808,-178.506,6.694,148.793
C02367=1163.506,152.075,-56.830,-178.503,6.696,148.793
C02368=1163.501,152.324,-56.850,-178.500,6.698,148.792
C02369=1163.496,152.573,-56.871,-178.498,6.700,148.792
C02370=1163.491,152.822,-56.893,-178.495,6.701,148.792
C02371=1163.486,153.071,-56.914,-178.492,6.703,148.791
C02372=1163.483,153.320,-56.935,-178.489,6.705,148.791
C02373=1163.477,153.569,-56.956,-178.487,6.707,148.790
C02374=1163.473,153.818,-56.978,-178.484,6.708,148.790
C02375=1163.467,154.067,-56.999,-178.481,6.710,148.790
C02376=1163.464,154.316,-57.020,-178.479,6.712,148.789
C02377=1163.459,154.566,-57.041,-178.476,6.713,148.789
C02378=1163.454,154.814,-57.063,-178.473,6.715,148.788
C02379=1163.449,155.063,-57.084,-178.471,6.717,148.788
C02380=1163.444,155.313,-57.106,-178.467,6.720,148.788
C02381=1163.440,155.562,-57.126,-178.465,6.721,148.787
C02382=1163.435,155.810,-57.148,-178.462,6.723,148.787
C02383=1163.430,156.059,-57.170,-178.459,6.725,148.787
C02384=1163.426,156.309,-57.191,-178.456,6.726,148.786
C02385=1163.421,156.558,-57.213,-178.454,6.728,148.786
C02386=1163.416,156.807,-57.234,-178.451,6.730,148.785
C02387=1163.411,157.056,-57.256,-178.448,6.732,148.785
C02388=1163.407,157.305,-57.277,-178.446,6.733,148.785
C02389=1163.402,157.554,-57.298,-178.443,6.736,148.785
C02390=1163.397,157.823,-57.322,-178.440,6.738,148.784
C02391=1163.392,158.092,-57.345,-178.437,6.740,148.784
C02392=1163.387,158.361,-57.368,-178.434,6.742,148.783
C02393=1163.382,158.629,-57.391,-178.431,6.744,148.783
C02394=1163.377,158.879,-57.412,-178.428,6.746,148.783
C02395=1163.372,159.127,-57.434,-178.426,6.747,148.782
C02396=1163.368,159.377,-57.456,-178.423,6.749,148.782
C02397=1163.363,159.626,-57.477,-178.420,6.751,148.781
C02398=1163.358,159.875,-57.499,-178.418,6.753,148.781
C02399=1163.354,160.124,-57.521,-178.415,6.755,148.781
C02400=1163.349,160.372,-57.543,-178.412,6.757,148.780
C02401=1163.344,160.622,-57.565,-178.409,6.759,148.780
C02402=1163.339,160.871,-57.586,-178.407,6.761,148.780
C02403=1163.334,161.120,-57.607,-178.404,6.762,148.779
C02404=1163.330,161.369,-57.629,-178.401,6.764,148.779
C02405=1163.325,161.618,-57.651,-178.399,6.766,148.779
C02406=1163.321,161.867,-57.673,-178.396,6.768,148.778
C02407=1163.316,162.116,-57.695,-178.393,6.770,148.778
C02408=1163.311,162.365,-57.716,-178.390,6.772,148.778
C02409=1163.307,162.614,-57.738,-178.388,6.774,148.777
C02410=1163.302,162.863,-57.759,-178.385,6.776,148.777
C02411=1163.297,163.112,-57.781,-178.382,6.778,148.777
C02412=1163.293,163.361,-57.803,-178.380,6.779,148.776
C02413=1163.288,163.610,-57.825,-178.377,6.781,148.776
C02414=1163.283,163.859,-57.847,-178.374,6.784,148.776
C02415=1163.279,164.108,-57.869,-178.371,6.785,148.775
C02416=1163.274,164.357,-57.891,-178.368,6.787,148.775
C02417=1163.269,164.606,-57.912,-178.366,6.789,148.774
C02418=1163.265,164.855,-57.934,-178.363,6.791,148.774
C02419=1163.260,165.103,-57.956,-178.361,6.793,148.774
C02420=1163.255,165.353,-57.979,-178.357,6.795,148.774
C02421=1163.250,165.602,-58.000,-178.355,6.797,148.773
C02422=1163.246,165.851,-58.022,-178.352,6.799,148.773
C02423=1163.241,166.100,-58.044,-178.349,6.801,148.772
C02424=1163.237,166.349,-58.066,-178.347,6.802,148.772
C02425=1163.232,166.598,-58.088,-178.344,6.804,148.772
C02426=1163.228,166.847,-58.110,-178.341,6.807,148.772
C02427=1163.222,167.096,-58.132,-178.338,6.809,148.771
C02428=1163.218,167.345,-58.154,-178.336,6.810,148.771
C02429=1163.213,167.594,-58.176,-178.333,6.812,148.770
C02430=1163.209,167.843,-58.199,-178.330,6.814,148.770
C02431=1163.204,168.091,-58.220,-178.328,6.816,148.770
C02432=1163.199,168.341,-58.243,-178.324,6.818,148.769
C02433=1163.194,168.590,-58.265,-178.322,6.820,148.769
C02434=1163.190,168.839,-58.287,-178.320,6.822,148.769
C02435=1163.185,169.088,-58.308,-178.317,6.824,148.768
C02436=1163.181,169.337,-58.332,-178.314,6.826,148.768
C02437=1163.176,169.585,-58.353,-178.311,6.828,148.768
C02438=1163.172,169.835,-58.375,-178.308,6.830,148.767
C02439=1163.167,170.083,-58.397,-178.306,6.832,148.767
C02440=1163.162,170.333,-58.420,-178.303,6.834,148.767
C02441=1163.157,170.581,-58.442,-178.301,6.836,148.766
C02442=1163.153,170.830,-58.464,-178.297,6.838,148.766
C02443=1163.149,171.080,-58.486,-178.295,6.840,148.766
C02444=1163.143,171.328,-58.509,-178.292,6.842,148.765
C02445=1163.139,171.577,-58.531,-178.289,6.843,148.765
C02446=1163.134,171.826,-58.553,-178.287,6.845,148.765
C02447=1163.129,172.076,-58.576,-178.284,6.848,148.765
C02448=1163.125,172.324,-58.598,-178.281,6.850,148.764
C02449=1163.120,172.573,-58.620,-178.278,6.852,148.764
C02450=1163.115,172.823,-58.643,-178.276,6.853,148.763
C02451=1163.111,173.071,-58.665,-178.273,6.855,148.763
C02452=1163.106,173.320,-58.687,-178.270,6.858,148.763
C02453=1163.102,173.569,-58.711,-178.268,6.860,148.763
C02454=1163.097,173.818,-58.732,-178.265,6.861,148.762
C02455=1163.092,174.067,-58.755,-178.262,6.863,148.762
C02456=1163.087,174.315,-58.777,-178.259,6.866,148.762
C02457=1163.083,174.565,-58.799,-178.257,6.868,148.761
C02458=1163.078,174.814,-58.823,-178.254,6.870,148.761
C02459=1163.073,175.062,-58.844,-178.251,6.871,148.761
C02460=1163.069,175.311,-58.868,-178.248,6.874,148.760
C02461=1163.064,175.561,-58.890,-178.245,6.876,148.760
C02462=1163.059,175.809,-58.913,-178.243,6.878,148.760
C02463=1163.055,176.058,-58.935,-178.240,6.880,148.759
C02464=1163.051,176.307,-58.958,-178.238,6.881,148.759
C02465=1163.045,176.556,-58.980,-178.235,6.884,148.759
C02466=1163.041,176.805,-59.003,-178.232,6.886,148.758
C02467=1163.036,177.054,-59.025,-178.230,6.888,148.758
C02468=1163.032,177.302,-59.048,-178.227,6.890,148.758
C02469=1163.027,177.552,-59.070,-178.224,6.892,148.758
C02470=1163.023,177.801,-59.093,-178.221,6.894,148.757
C02471=1163.018,178.050,-59.116,-178.218,6.896,148.757
C02472=1163.013,178.299,-59.138,-178.216,6.898,148.757
C02473=1163.009,178.548,-59.161,-178.213,6.900,148.756
C02474=1163.005,178.796,-59.184,-178.210,6.902,148.756
C02475=1163.000,179.046,-59.207,-178.207,6.904,148.756
C02476=1162.994,179.294,-59.230,-178.205,6.906,148.755
C02477=1162.990,179.543,-59.253,-178.202,6.908,148.755
C02478=1162.985,179.793,-59.275,-178.199,6.910,148.755
C02479=1162.981,180.041,-59.298,-178.197,6.912,148.754
C02480=1162.976,180.290,-59.321,-178.193,6.915,148.754
C02481=1162.972,180.539,-59.343,-178.191,6.917,148.754
C02482=1162.967,180.788,-59.366,-178.188,6.918,148.754
C02483=1162.962,181.037,-59.390,-178.186,6.920,148.753
C02484=1162.958,181.285,-59.412,-178.182,6.923,148.753
C02485=1162.953,181.535,-59.435,-178.180,6.925,148.753
C02486=1162.949,181.783,-59.458,-178.178,6.927,148.752
C02487=1162.944,182.033,-59.481,-178.174,6.929,148.752
C02488=1162.939,182.282,-59.504,-178.172,6.931,148.752
C02489=1162.935,182.530,-59.527,-178.169,6.933,148.751
C02490=1162.930,182.779,-59.549,-178.167,6.935,148.751
C02491=1162.925,183.028,-59.573,-178.163,6.937,148.751
C02492=1162.921,183.277,-59.595,-178.161,6.939,148.750
C02493=1162.917,183.526,-59.619,-178.159,6.941,148.750
C02494=1162.911,183.796,-59.644,-178.155,6.944,148.750
C02495=1162.907,184.065,-59.668,-178.153,6.946,148.750
C02496=1162.901,184.335,-59.693,-178.149,6.948,148.749
C02497=1162.896,184.604,-59.719,-178.146,6.951,148.749
C02498=1162.892,184.853,-59.741,-178.143,6.952,148.749
C02499=1162.887,185.103,-59.764,-178.141,6.955,148.748
C02500=1162.882,185.351,-59.787,-178.139,6.956,148.748
C02501=1162.877,185.600,-59.811,-178.135,6.959,148.748
C02502=1162.873,185.849,-59.834,-178.133,6.961,148.748
C02503=1162.869,186.098,-59.857,-178.130,6.963,148.747
C02504=1162.864,186.347,-59.880,-178.127,6.965,148.747
C02505=1162.859,186.596,-59.904,-178.124,6.967,148.747
C02506=1162.855,186.845,-59.927,-178.122,6.969,148.746
C02507=1162.851,187.093,-59.950,-178.119,6.972,148.746
C02508=1162.845,187.342,-59.973,-178.116,6.974,148.746
C02509=1162.841,187.591,-59.996,-178.114,6.976,148.746
C02510=1162.836,187.840,-60.020,-178.111,6.978,148.745
C02511=1162.832,188.088,-60.044,-178.108,6.980,148.745
C02512=1162.827,188.337,-60.067,-178.106,6.982,148.745
C02513=1162.823,188.586,-60.090,-178.103,6.985,148.744
C02514=1162.818,188.835,-60.113,-178.100,6.986,148.744
C02515=1162.813,189.084,-60.136,-178.097,6.988,148.744
C02516=1162.809,189.333,-60.160,-178.095,6.991,148.744
C02517=1162.804,189.582,-60.183,-178.092,6.993,148.743
C02518=1162.799,189.831,-60.207,-178.089,6.995,148.743
C02519=1162.795,190.080,-60.231,-178.086,6.998,148.743
C02520=1162.790,190.329,-60.254,-178.084,6.999,148.742
C02521=1162.786,190.578,-60.277,-178.081,7.001,148.742
C02522=1162.782,190.826,-60.300,-178.078,7.004,148.742
C02523=1162.777,191.075,-60.323,-178.076,7.006,148.742
C02524=1162.772,191.323,-60.347,-178.073,7.008,148.741
C02525=1162.767,191.572,-60.370,-178.070,7.011,148.741
C02526=1162.763,191.821,-60.394,-178.067,7.012,148.741
C02527=1162.758,192.070,-60.417,-178.065,7.014,148.740
C02528=1162.753,192.319,-60.441,-178.062,7.017,148.740
C02529=1162.749,192.568,-60.465,-178.059,7.019,148.740
C02530=1162.744,192.817,-60.488,-178.056,7.021,148.740
C02531=1162.740,193.065,-60.512,-178.054,7.023,148.740
C02532=1162.735,193.314,-60.535,-178.051,7.025,148.739
C02533=1162.731,193.564,-60.559,-178.048,7.028,148.739
C02534=1162.726,193.812,-60.583,-178.046,7.030,148.739
C02535=1162.722,194.061,-60.607,-178.043,7.032,148.738
C02536=1162.717,194.310,-60.630,-178.040,7.034,148.738
C02537=1162.713,194.559,-60.654,-178.038,7.036,148.738
C02538=1162.708,194.808,-60.677,-178.034,7.039,148.738
C02539=1162.704,195.056,-60.701,-178.032,7.041,148.737
C02540=1162.699,195.305,-60.725,-178.029,7.043,148.737
C02541=1162.694,195.554,-60.748,-178.026,7.045,148.737
C02542=1162.689,195.803,-60.773,-178.024,7.048,148.737
C02543=1162.684,196.052,-60.796,-178.021,7.049,148.736
C02544=1162.680,196.300,-60.820,-178.018,7.052,148.736
C02545=1162.675,196.549,-60.844,-178.016,7.054,148.736
C02546=1162.671,196.798,-60.868,-178.013,7.057,148.735
C02547=1162.666,197.047,-60.891,-178.010,7.058,148.735
C02548=1162.662,197.295,-60.915,-178.008,7.060,148.735
C02549=1162.658,197.545,-60.939,-178.004,7.063,148.735
C02550=1162.653,197.793,-60.963,-178.002,7.065,148.735
C02551=1162.648,198.043,-60.987,-177.999,7.068,148.734
C02552=1162.643,198.291,-61.011,-177.996,7.069,148.734
C02553=1162.639,198.540,-61.035,-177.994,7.072,148.734
C02554=1162.634,198.789,-61.058,-177.991,7.074,148.733
C02555=1162.630,199.037,-61.082,-177.988,7.076,148.733
C02556=1162.624,199.286,-61.106,-177.985,7.079,148.733
C02557=1162.621,199.536,-61.131,-177.983,7.081,148.733
C02558=1162.616,199.784,-61.155,-177.980,7.083,148.732
C02559=1162.612,200.033,-61.178,-177.977,7.085,148.732
C02560=1162.607,200.281,-61.202,-177.975,7.087,148.732
C02561=1162.602,200.530,-61.227,-177.972,7.090,148.732
C02562=1162.597,200.779,-61.250,-177.969,7.092,148.731
C02563=1162.594,201.028,-61.275,-177.966,7.095,148.731
C02564=1162.589,201.277,-61.299,-177.964,7.097,148.731
C02565=1162.584,201.525,-61.324,-177.961,7.098,148.731
C02566=1162.579,201.774,-61.347,-177.958,7.101,148.730
C02567=1162.575,202.023,-61.371,-177.955,7.103,148.730
C02568=1162.571,202.272,-61.395,-177.953,7.106,148.730
C02569=1162.566,202.521,-61.420,-177.950,7.108,148.730
C02570=1162.561,202.770,-61.443,-177.947,7.111,148.730
C02571=1162.557,203.018,-61.468,-177.945,7.112,148.729
C02572=1162.552,203.267,-61.492,-177.942,7.114,148.729
C02573=1162.548,203.516,-61.517,-177.939,7.117,148.729
C02574=1162.544,203.764,-61.541,-177.936,7.119,148.728
C02575=1162.538,204.014,-61.565,-177.934,7.122,148.728
C02576=1162.534,204.262,-61.589,-177.931,7.124,148.728
C02577=1162.530,204.511,-61.613,-177.928,7.126,148.728
C02578=1162.525,204.760,-61.638,-177.926,7.128,148.728
C02579=1162.520,205.008,-61.662,-177.922,7.131,148.727
C02580=1162.516,205.257,-61.686,-177.920,7.133,148.727
C02581=1162.512,205.506,-61.711,-177.917,7.135,148.727
C02582=1162.507,205.755,-61.735,-177.915,7.138,148.727
C02583=1162.502,206.003,-61.760,-177.912,7.139,148.726
C02584=1162.498,206.252,-61.784,-177.909,7.142,148.726
C02585=1162.493,206.501,-61.809,-177.906,7.144,148.726
C02586=1162.489,206.750,-61.833,-177.904,7.147,148.726
C02587=1162.484,206.998,-61.857,-177.901,7.149,148.725
C02588=1162.480,207.247,-61.882,-177.898,7.152,148.725
C02589=1162.475,207.496,-61.906,-177.896,7.154,148.725
C02590=1162.470,207.745,-61.931,-177.893,7.156,148.725
C02591=1162.466,207.994,-61.955,-177.890,7.158,148.725
C02592=1162.461,208.242,-61.980,-177.887,7.161,148.724
C02593=1162.457,208.491,-62.004,-177.885,7.163,148.724
C02594=1162.452,208.740,-62.029,-177.881,7.166,148.724
C02595=1162.448,208.989,-62.053,-177.879,7.168,148.724
C02596=1162.443,209.237,-62.078,-177.876,7.170,148.723
C02597=1162.439,209.487,-62.102,-177.874,7.172,148.723
C02598=1162.434,209.757,-62.129,-177.871,7.175,148.723
C02599=1162.429,210.027,-62.156,-177.868,7.178,148.723
C02600=1162.424,210.298,-62.183,-177.865,7.180,148.722
C02601=1162.419,210.568,-62.209,-177.862,7.182,148.722
C02602=1162.415,210.817,-62.235,-177.859,7.185,148.722
C02603=1162.409,211.066,-62.259,-177.856,7.187,148.722
C02604=1162.405,211.314,-62.283,-177.854,7.190,148.722
C02605=1162.401,211.563,-62.309,-177.851,7.192,148.721
C02606=1162.396,211.812,-62.333,-177.848,7.195,148.721
C02607=1162.392,212.061,-62.358,-177.845,7.196,148.721
C02608=1162.387,212.310,-62.383,-177.843,7.199,148.721
C02609=1162.383,212.558,-62.408,-177.840,7.201,148.720
C02610=1162.378,212.807,-62.433,-177.837,7.204,148.720
C02611=1162.374,213.055,-62.457,-177.835,7.206,148.720
C02612=1162.370,213.304,-62.482,-177.832,7.209,148.720
C02613=1162.364,213.553,-62.507,-177.829,7.211,148.720
C02614=1162.360,213.801,-62.531,-177.826,7.213,148.719
C02615=1162.356,214.050,-62.557,-177.824,7.215,148.719
C02616=1162.351,214.299,-62.582,-177.821,7.218,148.719
C02617=1162.347,214.548,-62.606,-177.818,7.220,148.719
C02618=1162.342,214.796,-62.631,-177.815,7.223,148.719
C02619=1162.337,215.046,-62.656,-177.813,7.225,148.718
C02620=1162.332,215.294,-62.681,-177.810,7.228,148.718
C02621=1162.329,215.543,-62.706,-177.808,7.230,148.718
C02622=1162.324,215.792,-62.731,-177.805,7.232,148.718
C02623=1162.319,216.040,-62.757,-177.802,7.234,148.718
C02624=1162.315,216.289,-62.781,-177.799,7.237,148.717
C02625=1162.311,216.538,-62.807,-177.796,7.240,148.717
C02626=1162.306,216.786,-62.831,-177.794,7.242,148.717
C02627=1162.302,217.035,-62.857,-177.791,7.245,148.717
C02628=1162.296,217.284,-62.882,-177.788,7.246,148.716
C02629=1162.293,217.532,-62.907,-177.785,7.249,148.716
C02630=1162.288,217.781,-62.931,-177.783,7.252,148.716
C02631=1162.284,218.030,-62.957,-177.780,7.254,148.716
C02632=1162.278,218.279,-62.982,-177.778,7.256,148.716
C02633=1162.274,218.527,-63.008,-177.775,7.259,148.715
C02634=1162.270,218.776,-63.032,-177.772,7.261,148.715
C02635=1162.266,219.025,-63.057,-177.769,7.264,148.715
C02636=1162.261,219.273,-63.083,-177.766,7.266,148.715
C02637=1162.256,219.522,-63.108,-177.764,7.268,148.715
C02638=1162.252,219.771,-63.134,-177.761,7.271,148.715
C02639=1162.247,220.019,-63.159,-177.759,7.273,148.714
C02640=1162.243,220.268,-63.183,-177.755,7.276,148.714
C02641=1162.239,220.516,-63.209,-177.753,7.278,148.714
C02642=1162.234,220.765,-63.235,-177.750,7.281,148.714
C02643=1162.229,221.014,-63.259,-177.747,7.284,148.714
C02644=1162.225,221.263,-63.285,-177.745,7.286,148.713
C02645=1162.221,221.511,-63.311,-177.742,7.288,148.713
C02646=1162.216,221.760,-63.335,-177.740,7.290,148.713
C02647=1162.211,222.009,-63.361,-177.736,7.293,148.713
C02648=1162.207,222.257,-63.387,-177.734,7.295,148.713
C02649=1162.202,222.506,-63.412,-177.731,7.298,148.713
C02650=1162.198,222.755,-63.437,-177.728,7.301,148.712
C02651=1162.193,223.003,-63.463,-177.726,7.303,148.712
C02652=1162.189,223.252,-63.488,-177.723,7.305,148.712
C02653=1162.185,223.501,-63.514,-177.721,7.308,148.712
C02654=1162.180,223.749,-63.540,-177.718,7.310,148.712
C02655=1162.175,223.998,-63.565,-177.715,7.313,148.711
C02656=1162.171,224.247,-63.590,-177.712,7.315,148.711
C02657=1162.166,224.495,-63.616,-177.709,7.318,148.711
C02658=1162.162,224.744,-63.642,-177.707,7.320,148.711
C02659=1162.158,224.993,-63.667,-177.704,7.323,148.711
C02660=1162.153,225.241,-63.693,-177.701,7.325,148.710
C02661=1162.149,225.490,-63.718,-177.699,7.328,148.710
C02662=1162.144,225.739,-63.744,-177.696,7.330,148.710
C02663=1162.140,225.987,-63.770,-177.693,7.332,148.710
C02664=1162.135,226.236,-63.795,-177.690,7.335,148.710
C02665=1162.131,226.484,-63.821,-177.687,7.338,148.709
C02666=1162.126,226.732,-63.846,-177.685,7.340,148.709
C02667=1162.122,226.981,-63.872,-177.682,7.343,148.709
C02668=1162.118,227.230,-63.898,-177.679,7.345,148.709
C02669=1162.112,227.479,-63.924,-177.677,7.348,148.709
C02670=1162.108,227.727,-63.950,-177.674,7.351,148.709
C02671=1162.104,227.976,-63.975,-177.671,7.352,148.708
C02672=1162.100,228.225,-64.001,-177.669,7.355,148.708
C02673=1162.095,228.473,-64.027,-177.666,7.358,148.708
C02674=1162.091,228.722,-64.052,-177.663,7.360,148.708
C02675=1162.086,228.971,-64.078,-177.660,7.363,148.708
C02676=1162.081,229.220,-64.104,-177.658,7.366,148.708
C02677=1162.077,229.468,-64.130,-177.655,7.368,148.707
C02678=1162.072,229.717,-64.156,-177.652,7.371,148.707
C02679=1162.068,229.965,-64.182,-177.649,7.374,148.707
C02680=1162.064,230.214,-64.208,-177.647,7.375,148.707
C02681=1162.059,230.463,-64.234,-177.644,7.378,148.707
C02682=1162.054,230.711,-64.259,-177.641,7.381,148.707
C02683=1162.050,230.960,-64.285,-177.639,7.383,148.706
C02684=1162.046,231.208,-64.312,-177.636,7.386,148.706
C02685=1162.041,231.457,-64.338,-177.634,7.388,148.706
C02686=1162.036,231.705,-64.363,-177.630,7.391,148.706
C02687=1162.032,231.954,-64.389,-177.628,7.394,148.706
C02688=1162.028,232.203,-64.415,-177.625,7.396,148.706
C02689=1162.023,232.451,-64.442,-177.622,7.398,148.705
C02690=1162.019,232.700,-64.468,-177.619,7.401,148.705
C02691=1162.015,232.949,-64.494,-177.617,7.403,148.705
C02692=1162.010,233.197,-64.520,-177.614,7.406,148.705
C02693=1162.005,233.445,-64.546,-177.611,7.409,148.705
C02694=1162.001,233.694,-64.572,-177.609,7.411,148.705
C02695=1161.997,233.943,-64.599,-177.606,7.414,148.705
C02696=1161.992,234.191,-64.625,-177.603,7.417,148.704
C02697=1161.988,234.440,-64.650,-177.600,7.420,148.704
C02698=1161.983,234.689,-64.677,-177.598,7.422,148.704
C02699=1161.979,234.937,-64.703,-177.595,7.424,148.704
C02700=1161.975,235.185,-64.729,-177.592,7.427,148.704
C02701=1161.970,235.434,-64.756,-177.590,7.429,148.704
C02702=1161.965,235.705,-64.784,-177.587,7.432,148.704
C02703=1161.960,235.978,-64.813,-177.584,7.435,148.703
C02704=1161.956,236.249,-64.842,-177.581,7.438,148.703
C02705=1161.950,236.521,-64.870,-177.578,7.440,148.703
C02706=1161.946,236.769,-64.897,-177.575,7.443,148.703
C02707=1161.941,237.019,-64.923,-177.572,7.446,148.703
C02708=1161.937,237.267,-64.950,-177.570,7.448,148.703
C02709=1161.933,237.515,-64.975,-177.567,7.451,148.702
C02710=1161.928,237.764,-65.002,-177.564,7.454,148.702
C02711=1161.924,238.013,-65.028,-177.561,7.457,148.702
C02712=1161.920,238.261,-65.055,-177.559,7.459,148.702
C02713=1161.916,238.509,-65.082,-177.556,7.462,148.702
C02714=1161.911,238.759,-65.108,-177.553,7.465,148.702
C02715=1161.907,239.007,-65.134,-177.551,7.467,148.702
C02716=1161.902,239.256,-65.161,-177.548,7.470,148.702
C02717=1161.898,239.504,-65.187,-177.545,7.472,148.701
C02718=1161.893,239.753,-65.214,-177.542,7.475,148.701
C02719=1161.888,240.001,-65.240,-177.540,7.477,148.701
C02720=1161.884,240.249,-65.267,-177.537,7.480,148.701
C02721=1161.879,240.498,-65.294,-177.534,7.483,148.701
C02722=1161.875,240.746,-65.320,-177.532,7.485,148.701
C02723=1161.870,240.995,-65.347,-177.529,7.488,148.701
C02724=1161.866,241.243,-65.373,-177.526,7.491,148.701
C02725=1161.862,241.492,-65.400,-177.523,7.494,148.701
C02726=1161.857,241.741,-65.427,-177.521,7.496,148.700
C02727=1161.853,241.990,-65.453,-177.518,7.499,148.700
C02728=1161.849,242.238,-65.480,-177.515,7.502,148.700
C02729=1161.845,242.486,-65.507,-177.512,7.505,148.700
C02730=1161.840,242.735,-65.534,-177.510,7.507,148.700
C02731=1161.835,242.984,-65.560,-177.507,7.509,148.700
C02732=1161.831,243.232,-65.587,-177.504,7.512,148.700
C02733=1161.827,243.481,-65.614,-177.501,7.515,148.699
C02734=1161.822,243.729,-65.641,-177.499,7.517,148.699
C02735=1161.818,243.977,-65.667,-177.497,7.520,148.699
C02736=1161.813,244.226,-65.694,-177.493,7.523,148.699
C02737=1161.809,244.474,-65.722,-177.491,7.526,148.699
C02738=1161.804,244.723,-65.747,-177.488,7.528,148.699
C02739=1161.800,244.972,-65.774,-177.486,7.531,148.699
C02740=1161.795,245.220,-65.801,-177.483,7.534,148.699
C02741=1161.790,245.469,-65.828,-177.480,7.537,148.699
C02742=1161.787,245.717,-65.855,-177.477,7.539,148.698
C02743=1161.782,245.966,-65.882,-177.475,7.542,148.698
C02744=1161.778,246.214,-65.909,-177.472,7.544,148.698
C02745=1161.773,246.463,-65.936,-177.469,7.547,148.698
C02746=1161.769,246.711,-65.963,-177.467,7.550,148.698
C02747=1161.765,246.960,-65.990,-177.464,7.552,148.698
C02748=1161.760,247.208,-66.017,-177.461,7.555,148.698
C02749=1161.755,247.457,-66.044,-177.458,7.558,148.698
C02750=1161.751,247.705,-66.071,-177.456,7.560,148.697
C02751=1161.747,247.954,-66.098,-177.453,7.563,148.697
C02752=1161.743,248.202,-66.126,-177.450,7.566,148.697
C02753=1161.738,248.450,-66.153,-177.448,7.569,148.697
C02754=1161.734,248.699,-66.180,-177.445,7.572,148.697
C02755=1161.729,248.947,-66.207,-177.443,7.574,148.697
C02756=1161.724,249.196,-66.234,-177.439,7.577,148.697
C02757=1161.721,249.445,-66.261,-177.437,7.580,148.697
C02758=1161.716,249.693,-66.288,-177.434,7.583,148.697
C02759=1161.712,249.941,-66.316,-177.432,7.585,148.697
C02760=1161.707,250.190,-66.343,-177.429,7.588,148.697
C02761=1161.703,250.438,-66.370,-177.426,7.591,148.696
C02762=1161.699,250.687,-66.397,-177.423,7.594,148.696
C02763=1161.694,250.936,-66.424,-177.421,7.597,148.696
C02764=1161.690,251.184,-66.452,-177.418,7.598,148.696
C02765=1161.685,251.432,-66.479,-177.415,7.601,148.696
C02766=1161.680,251.681,-66.506,-177.412,7.604,148.696
C02767=1161.676,251.930,-66.534,-177.410,7.607,148.696
C02768=1161.672,252.178,-66.561,-177.407,7.610,148.696
C02769=1161.668,252.426,-66.588,-177.405,7.612,148.696
C02770=1161.663,252.674,-66.615,-177.402,7.615,148.696
C02771=1161.660,252.923,-66.643,-177.399,7.618,148.696
C02772=1161.655,253.171,-66.670,-177.396,7.621,148.695
C02773=1161.650,253.420,-66.697,-177.394,7.624,148.695
C02774=1161.646,253.668,-66.725,-177.391,7.627,148.695
C02775=1161.642,253.917,-66.752,-177.388,7.629,148.695
C02776=1161.638,254.165,-66.780,-177.386,7.632,148.695
C02777=1161.633,254.413,-66.807,-177.383,7.635,148.695
C02778=1161.628,254.663,-66.835,-177.380,7.638,148.695
C02779=1161.624,254.911,-66.863,-177.377,7.641,148.695
C02780=1161.619,255.159,-66.890,-177.375,7.643,148.695
C02781=1161.615,255.407,-66.918,-177.372,7.646,148.695
C02782=1161.611,255.656,-66.945,-177.370,7.649,148.695
C02783=1161.606,255.904,-66.973,-177.367,7.652,148.694
C02784=1161.602,256.153,-67.000,-177.364,7.655,148.694
C02785=1161.598,256.401,-67.028,-177.361,7.657,148.694
C02786=1161.593,256.650,-67.055,-177.359,7.660,148.694
C02787=1161.589,256.898,-67.083,-177.356,7.663,148.694
C02788=1161.585,257.147,-67.111,-177.354,7.665,148.694
C02789=1161.580,257.395,-67.139,-177.351,7.668,148.694
C02790=1161.575,257.643,-67.167,-177.348,7.671,148.694
C02791=1161.571,257.892,-67.194,-177.345,7.674,148.694
C02792=1161.567,258.140,-67.222,-177.343,7.676,148.694
C02793=1161.563,258.389,-67.249,-177.340,7.679,148.694
C02794=1161.559,258.637,-67.277,-177.338,7.682,148.694
C02795=1161.553,258.885,-67.305,-177.335,7.685,148.694
C02796=1161.549,259.134,-67.333,-177.332,7.688,148.693
C02797=1161.545,259.382,-67.361,-177.329,7.691,148.693
C02798=1161.541,259.630,-67.388,-177.326,7.694,148.693
C02799=1161.537,259.879,-67.416,-177.324,7.696,148.693
C02800=1161.532,260.128,-67.444,-177.321,7.699,148.693
C02801=1161.528,260.376,-67.472,-177.318,7.702,148.693
C02802=1161.523,260.624,-67.500,-177.316,7.705,148.693
C02803=1161.519,260.873,-67.528,-177.313,7.708,148.693
C02804=1161.514,261.121,-67.556,-177.310,7.711,148.693
C02805=1161.510,261.369,-67.584,-177.307,7.714,148.693
C02806=1161.505,261.643,-67.614,-177.304,7.717,148.693
C02807=1161.501,261.916,-67.645,-177.302,7.720,148.693
C02808=1161.496,262.189,-67.676,-177.299,7.723,148.693
C02809=1161.491,262.463,-67.706,-177.296,7.726,148.693
C02810=1161.486,262.711,-67.735,-177.293,7.728,148.693
C02811=1161.482,262.959,-67.763,-177.291,7.731,148.692
C02812=1161.478,263.207,-67.791,-177.288,7.734,148.692
C02813=1161.474,263.456,-67.820,-177.285,7.737,148.692
C02814=1161.469,263.704,-67.847,-177.282,7.740,148.692
C02815=1161.466,263.953,-67.875,-177.280,7.743,148.692
C02816=1161.460,264.201,-67.904,-177.277,7.746,148.692
C02817=1161.457,264.449,-67.932,-177.274,7.749,148.692
C02818=1161.452,264.698,-67.960,-177.272,7.751,148.692
C02819=1161.448,264.946,-67.988,-177.269,7.754,148.692
C02820=1161.444,265.194,-68.016,-177.266,7.757,148.692
C02821=1161.439,265.443,-68.045,-177.264,7.760,148.692
C02822=1161.435,265.691,-68.073,-177.261,7.763,148.692
C02823=1161.430,265.940,-68.101,-177.259,7.766,148.692
C02824=1161.426,266.188,-68.129,-177.256,7.769,148.692
C02825=1161.421,266.436,-68.158,-177.253,7.772,148.692
C02826=1161.417,266.684,-68.186,-177.250,7.775,148.692
C02827=1161.413,266.933,-68.215,-177.248,7.777,148.692
C02828=1161.408,267.181,-68.242,-177.245,7.780,148.692
C02829=1161.404,267.430,-68.270,-177.243,7.783,148.692
C02830=1161.400,267.679,-68.299,-177.240,7.786,148.692
C02831=1161.396,267.926,-68.327,-177.237,7.789,148.692
C02832=1161.391,268.175,-68.356,-177.234,7.792,148.691
C02833=1161.386,268.423,-68.385,-177.232,7.795,148.691
C02834=1161.383,268.671,-68.413,-177.229,7.798,148.691
C02835=1161.377,268.920,-68.441,-177.226,7.801,148.692
C02836=1161.374,269.168,-68.469,-177.224,7.804,148.691
C02837=1161.369,269.417,-68.498,-177.222,7.806,148.691
C02838=1161.365,269.664,-68.527,-177.219,7.809,148.691
C02839=1161.361,269.913,-68.555,-177.216,7.812,148.691
C02840=1161.356,270.161,-68.583,-177.213,7.815,148.691
C02841=1161.352,270.410,-68.612,-177.210,7.818,148.691
C02842=1161.348,270.658,-68.641,-177.208,7.821,148.691
C02843=1161.343,270.906,-68.669,-177.205,7.824,148.691
C02844=1161.339,271.155,-68.698,-177.202,7.827,148.691
C02845=1161.335,271.404,-68.726,-177.200,7.830,148.691
C02846=1161.330,271.651,-68.755,-177.197,7.833,148.691
C02847=1161.326,271.900,-68.784,-177.194,7.836,148.691
C02848=1161.322,272.149,-68.812,-177.192,7.839,148.691
C02849=1161.317,272.396,-68.841,-177.189,7.842,148.691
C02850=1161.313,272.645,-68.870,-177.187,7.844,148.691
C02851=1161.309,272.893,-68.899,-177.184,7.847,148.691
C02852=1161.304,273.141,-68.927,-177.182,7.851,148.691
C02853=1161.300,273.390,-68.956,-177.179,7.853,148.691
C02854=1161.296,273.638,-68.985,-177.176,7.856,148.691
C02855=1161.291,273.886,-69.013,-177.173,7.859,148.691
C02856=1161.287,274.135,-69.042,-177.171,7.862,148.691
C02857=1161.283,274.383,-69.071,-177.168,7.865,148.691
C02858=1161.279,274.631,-69.100,-177.165,7.868,148.691
C02859=1161.274,274.880,-69.128,-177.163,7.872,148.691
C02860=1161.270,275.128,-69.158,-177.160,7.875,148.691
C02861=1161.266,275.376,-69.186,-177.157,7.877,148.691
C02862=1161.261,275.624,-69.215,-177.154,7.880,148.691
C02863=1161.257,275.873,-69.244,-177.152,7.883,148.691
C02864=1161.253,276.121,-69.273,-177.149,7.886,148.691
C02865=1161.248,276.369,-69.303,-177.147,7.890,148.691
C02866=1161.244,276.617,-69.331,-177.144,7.893,148.691
C02867=1161.240,276.866,-69.360,-177.141,7.896,148.691
C02868=1161.235,277.114,-69.389,-177.139,7.898,148.691
C02869=1161.231,277.363,-69.418,-177.136,7.901,148.691
C02870=1161.227,277.610,-69.447,-177.134,7.904,148.691
C02871=1161.223,277.859,-69.475,-177.131,7.907,148.691
C02872=1161.219,278.107,-69.505,-177.128,7.910,148.691
C02873=1161.214,278.355,-69.534,-177.126,7.913,148.691
C02874=1161.210,278.604,-69.564,-177.123,7.916,148.691
C02875=1161.205,278.852,-69.592,-177.120,7.919,148.691
C02876=1161.201,279.100,-69.622,-177.118,7.922,148.691
C02877=1161.197,279.348,-69.651,-177.115,7.925,148.691
C02878=1161.192,279.597,-69.680,-177.112,7.928,148.691
C02879=1161.189,279.845,-69.709,-177.110,7.931,148.691
C02880=1161.185,280.093,-69.738,-177.107,7.934,148.691
C02881=1161.180,280.341,-69.767,-177.104,7.937,148.691
C02882=1161.176,280.589,-69.797,-177.102,7.940,148.691
C02883=1161.171,280.838,-69.825,-177.099,7.943,148.691
C02884=1161.167,281.086,-69.855,-177.096,7.946,148.691
C02885=1161.163,281.335,-69.884,-177.094,7.949,148.691
C02886=1161.159,281.583,-69.914,-177.091,7.952,148.691
C02887=1161.154,281.831,-69.943,-177.088,7.955,148.691
C02888=1161.150,282.079,-69.972,-177.086,7.958,148.691
C02889=1161.146,282.327,-70.002,-177.083,7.961,148.691
C02890=1161.141,282.575,-70.031,-177.081,7.964,148.691
C02891=1161.137,282.824,-70.061,-177.078,7.967,148.691
C02892=1161.133,283.072,-70.090,-177.075,7.970,148.691
C02893=1161.128,283.321,-70.119,-177.073,7.974,148.691
C02894=1161.124,283.569,-70.148,-177.070,7.977,148.691
C02895=1161.120,283.817,-70.178,-177.067,7.979,148.691
C02896=1161.115,284.065,-70.207,-177.064,7.982,148.691
C02897=1161.111,284.313,-70.236,-177.062,7.986,148.691
C02898=1161.106,284.562,-70.266,-177.059,7.989,148.691
C02899=1161.102,284.809,-70.297,-177.057,7.992,148.691
C02900=1161.098,285.058,-70.326,-177.054,7.995,148.691
C02901=1161.094,285.306,-70.355,-177.052,7.998,148.691
C02902=1161.090,285.554,-70.385,-177.049,8.001,148.691
C02903=1161.086,285.802,-70.414,-177.046,8.004,148.691
C02904=1161.081,286.051,-70.444,-177.044,8.007,148.691
C02905=1161.077,286.299,-70.473,-177.041,8.010,148.691
C02906=1161.072,286.548,-70.503,-177.038,8.013,148.691
C02907=1161.068,286.796,-70.533,-177.036,8.016,148.691
C02908=1161.064,287.044,-70.562,-177.033,8.019,148.691
C02909=1161.060,287.292,-70.592,-177.030,8.022,148.691
C02910=1161.055,287.567,-70.625,-177.028,8.025,148.691
C02911=1161.051,287.842,-70.658,-177.025,8.029,148.691
C02912=1161.046,288.117,-70.691,-177.022,8.032,148.691
C02913=1161.041,288.392,-70.724,-177.019,8.036,148.691
C02914=1161.037,288.640,-70.754,-177.016,8.039,148.691
C02915=1161.033,288.889,-70.783,-177.014,8.042,148.691
C02916=1161.029,289.136,-70.813,-177.011,8.045,148.691
C02917=1161.024,289.385,-70.843,-177.008,8.048,148.691
C02918=1161.020,289.633,-70.873,-177.006,8.051,148.691
C02919=1161.015,289.881,-70.902,-177.003,8.054,148.691
C02920=1161.012,290.129,-70.932,-177.000,8.057,148.691
C02921=1161.007,290.378,-70.962,-176.998,8.061,148.692
C02922=1161.002,290.626,-70.992,-176.995,8.064,148.692
C02923=1160.999,290.873,-71.022,-176.993,8.067,148.691
C02924=1160.994,291.122,-71.052,-176.990,8.070,148.692
C02925=1160.990,291.370,-71.082,-176.987,8.073,148.692
C02926=1160.986,291.618,-71.112,-176.985,8.076,148.692
C02927=1160.981,291.867,-71.142,-176.982,8.079,148.692
C02928=1160.977,292.115,-71.172,-176.980,8.082,148.692
C02929=1160.973,292.363,-71.202,-176.977,8.085,148.692
C02930=1160.969,292.611,-71.233,-176.975,8.088,148.692
C02931=1160.964,292.859,-71.262,-176.972,8.091,148.692
C02932=1160.961,293.107,-71.292,-176.970,8.095,148.692
C02933=1160.956,293.356,-71.322,-176.966,8.098,148.692
C02934=1160.952,293.603,-71.352,-176.963,8.101,148.692
C02935=1160.948,293.852,-71.382,-176.961,8.105,148.692
C02936=1160.943,294.099,-71.413,-176.958,8.107,148.692
C02937=1160.939,294.348,-71.442,-176.956,8.110,148.692
C02938=1160.935,294.596,-71.473,-176.953,8.114,148.692
C02939=1160.931,294.844,-71.503,-176.951,8.117,148.692
C02940=1160.926,295.093,-71.533,-176.948,8.120,148.692
C02941=1160.922,295.340,-71.564,-176.946,8.123,148.692
C02942=1160.918,295.588,-71.594,-176.943,8.126,148.692
C02943=1160.913,295.837,-71.624,-176.941,8.129,148.693
C02944=1160.910,296.085,-71.654,-176.938,8.132,148.692
C02945=1160.905,296.333,-71.685,-176.935,8.135,148.693
C02946=1160.901,296.581,-71.715,-176.933,8.138,148.693
C02947=1160.897,296.829,-71.745,-176.930,8.141,148.693
C02948=1160.893,297.077,-71.775,-176.928,8.145,148.693
C02949=1160.888,297.326,-71.806,-176.925,8.148,148.693
C02950=1160.885,297.574,-71.836,-176.922,8.152,148.693
C02951=1160.880,297.822,-71.867,-176.919,8.155,148.693
C02952=1160.875,298.070,-71.898,-176.917,8.158,148.693
C02953=1160.871,298.318,-71.927,-176.914,8.161,148.693
C02954=1160.867,298.566,-71.958,-176.911,8.164,148.693
C02955=1160.863,298.814,-71.988,-176.909,8.167,148.693
C02956=1160.859,299.062,-72.019,-176.906,8.170,148.693
C02957=1160.855,299.310,-72.049,-176.904,8.173,148.693
C02958=1160.850,299.559,-72.080,-176.901,8.176,148.693
C02959=1160.846,299.807,-72.110,-176.899,8.180,148.694
C02960=1160.842,300.055,-72.141,-176.896,8.183,148.694
C02961=1160.837,300.303,-72.171,-176.894,8.186,148.694
C02962=1160.833,300.551,-72.202,-176.891,8.190,148.694
C02963=1160.829,300.799,-72.233,-176.888,8.193,148.694
C02964=1160.825,301.047,-72.263,-176.886,8.196,148.694
C02965=1160.821,301.294,-72.294,-176.883,8.199,148.694
C02966=1160.817,301.543,-72.325,-176.881,8.202,148.694
C02967=1160.812,301.791,-72.355,-176.878,8.205,148.694
C02968=1160.808,302.039,-72.386,-176.876,8.208,148.694
C02969=1160.804,302.287,-72.417,-176.873,8.211,148.694
C02970=1160.800,302.535,-72.448,-176.870,8.215,148.694
C02971=1160.795,302.783,-72.478,-176.868,8.218,148.694
C02972=1160.791,303.031,-72.508,-176.865,8.222,148.695
C02973=1160.787,303.280,-72.540,-176.862,8.225,148.694
C02974=1160.783,303.528,-72.570,-176.860,8.228,148.695
C02975=1160.778,303.776,-72.601,-176.857,8.231,148.695
C02976=1160.775,304.024,-72.632,-176.855,8.234,148.695
C02977=1160.770,304.272,-72.662,-176.852,8.237,148.695
C02978=1160.766,304.520,-72.693,-176.850,8.240,148.695
C02979=1160.762,304.768,-72.724,-176.847,8.243,148.695
C02980=1160.757,305.016,-72.756,-176.845,8.247,148.695
C02981=1160.753,305.263,-72.786,-176.841,8.251,148.695
C02982=1160.749,305.512,-72.817,-176.839,8.254,148.695
C02983=1160.745,305.760,-72.848,-176.836,8.257,148.695
C02984=1160.741,306.009,-72.879,-176.834,8.260,148.695
C02985=1160.736,306.257,-72.910,-176.831,8.263,148.695
C02986=1160.732,306.504,-72.941,-176.829,8.266,148.696
C02987=1160.728,306.753,-72.972,-176.826,8.269,148.696
C02988=1160.724,307.000,-73.003,-176.824,8.273,148.696
C02989=1160.719,307.248,-73.033,-176.821,8.277,148.696
C02990=1160.716,307.496,-73.065,-176.818,8.280,148.696
C02991=1160.711,307.744,-73.096,-176.816,8.283,148.696
C02992=1160.707,307.993,-73.127,-176.813,8.286,148.696
C02993=1160.703,308.240,-73.159,-176.811,8.289,148.696
C02994=1160.699,308.489,-73.190,-176.808,8.292,148.696
C02995=1160.694,308.737,-73.220,-176.806,8.295,148.697
C02996=1160.690,308.984,-73.252,-176.803,8.298,148.697
C02997=1160.686,309.233,-73.283,-176.800,8.302,148.697
C02998=1160.681,309.481,-73.314,-176.798,8.306,148.697
C02999=1160.677,309.729,-73.346,-176.795,8.309,148.697
C03000=1160.674,309.977,-73.376,-176.793,8.312,148.697
C03001=1160.670,310.225,-73.408,-176.790,8.315,148.697
C03002=1160.665,310.473,-73.438,-176.788,8.318,148.697
C03003=1160.662,310.721,-73.470,-176.785,8.321,148.697
C03004=1160.657,310.969,-73.501,-176.782,8.325,148.697
C03005=1160.653,311.217,-73.533,-176.780,8.329,148.698
C03006=1160.649,311.465,-73.564,-176.777,8.332,148.698
C03007=1160.644,311.713,-73.596,-176.775,8.335,148.698
C03008=1160.640,311.961,-73.627,-176.772,8.338,148.698
C03009=1160.636,312.209,-73.659,-176.770,8.341,148.698
C03010=1160.631,312.457,-73.689,-176.767,8.345,148.698
C03011=1160.628,312.705,-73.721,-176.764,8.348,148.698
C03012=1160.623,312.953,-73.752,-176.762,8.351,148.698
C03013=1160.619,313.201,-73.784,-176.759,8.354,148.698
C03014=1160.614,313.478,-73.819,-176.756,8.359,148.699
C03015=1160.610,313.755,-73.855,-176.754,8.362,148.699
C03016=1160.605,314.033,-73.889,-176.751,8.366,148.699
C03017=1160.600,314.309,-73.925,-176.748,8.370,148.699
C03018=1160.596,314.558,-73.956,-176.745,8.373,148.699
C03019=1160.592,314.806,-73.988,-176.743,8.376,148.699
C03020=1160.588,315.054,-74.019,-176.740,8.379,148.699
C03021=1160.584,315.302,-74.051,-176.738,8.382,148.699
C03022=1160.580,315.549,-74.082,-176.735,8.386,148.700
C03023=1160.576,315.798,-74.113,-176.732,8.390,148.700
C03024=1160.571,316.045,-74.145,-176.730,8.393,148.700
C03025=1160.567,316.293,-74.177,-176.727,8.396,148.700
C03026=1160.563,316.541,-74.209,-176.725,8.399,148.700
C03027=1160.559,316.789,-74.241,-176.722,8.402,148.700
C03028=1160.555,317.037,-74.272,-176.719,8.406,148.700
C03029=1160.551,317.286,-74.304,-176.717,8.409,148.700
C03030=1160.546,317.533,-74.336,-176.714,8.412,148.701
C03031=1160.543,317.781,-74.368,-176.712,8.416,148.701
C03032=1160.538,318.028,-74.399,-176.709,8.419,148.701
C03033=1160.534,318.277,-74.431,-176.706,8.423,148.701
C03034=1160.530,318.525,-74.463,-176.704,8.426,148.701
C03035=1160.526,318.772,-74.495,-176.702,8.429,148.701
C03036=1160.522,319.021,-74.526,-176.699,8.432,148.701
C03037=1160.517,319.269,-74.558,-176.697,8.436,148.702
C03038=1160.513,319.516,-74.590,-176.694,8.440,148.702
C03039=1160.509,319.764,-74.622,-176.691,8.443,148.702
C03040=1160.505,320.013,-74.654,-176.689,8.446,148.702
C03041=1160.501,320.260,-74.686,-176.687,8.449,148.702
C03042=1160.497,320.508,-74.717,-176.684,8.452,148.702
C03043=1160.492,320.757,-74.750,-176.681,8.456,148.702
C03044=1160.489,321.005,-74.782,-176.679,8.460,148.703
C03045=1160.484,321.252,-74.813,-176.676,8.463,148.703
C03046=1160.480,321.500,-74.846,-176.674,8.466,148.703
C03047=1160.477,321.748,-74.878,-176.671,8.469,148.703
C03048=1160.472,321.995,-74.910,-176.668,8.473,148.703
C03049=1160.468,322.243,-74.942,-176.666,8.476,148.703
C03050=1160.464,322.491,-74.974,-176.663,8.480,148.703
C03051=1160.460,322.740,-75.006,-176.661,8.483,148.704
C03052=1160.455,322.987,-75.038,-176.659,8.486,148.704
C03053=1160.452,323.235,-75.070,-176.655,8.490,148.704
C03054=1160.447,323.483,-75.103,-176.653,8.493,148.704
C03055=1160.444,323.731,-75.135,-176.651,8.497,148.704
C03056=1160.439,323.979,-75.167,-176.648,8.500,148.704
C03057=1160.435,324.227,-75.199,-176.645,8.504,148.704
C03058=1160.431,324.475,-75.231,-176.643,8.507,148.705
C03059=1160.427,324.722,-75.264,-176.641,8.510,148.705
C03060=1160.423,324.971,-75.296,-176.638,8.513,148.705
C03061=1160.418,325.218,-75.328,-176.636,8.517,148.705
C03062=1160.414,325.466,-75.361,-176.633,8.521,148.705
C03063=1160.411,325.714,-75.393,-176.630,8.524,148.705
C03064=1160.406,325.962,-75.425,-176.628,8.527,148.706
C03065=1160.402,326.210,-75.457,-176.626,8.530,148.706
C03066=1160.398,326.457,-75.490,-176.622,8.534,148.706
C03067=1160.394,326.705,-75.522,-176.620,8.537,148.706
C03068=1160.390,326.953,-75.555,-176.618,8.541,148.706
C03069=1160.386,327.201,-75.587,-176.615,8.544,148.706
C03070=1160.382,327.449,-75.619,-176.613,8.548,148.707
C03071=1160.378,327.697,-75.652,-176.610,8.551,148.707
C03072=1160.373,327.944,-75.684,-176.608,8.554,148.707
C03073=1160.369,328.192,-75.717,-176.605,8.558,148.707
C03074=1160.365,328.440,-75.749,-176.602,8.562,148.707
C03075=1160.361,328.688,-75.782,-176.600,8.565,148.708
C03076=1160.357,328.936,-75.814,-176.598,8.568,148.708
C03077=1160.353,329.184,-75.847,-176.595,8.571,148.708
C03078=1160.349,329.432,-75.879,-176.592,8.575,148.708
C03079=1160.344,329.679,-75.912,-176.590,8.579,148.708
C03080=1160.341,329.927,-75.944,-176.588,8.582,148.708
C03081=1160.336,330.175,-75.977,-176.585,8.585,148.709
C03082=1160.332,330.423,-76.009,-176.582,8.589,148.709
C03083=1160.329,330.671,-76.042,-176.580,8.592,148.709
C03084=1160.324,330.919,-76.074,-176.577,8.596,148.709
C03085=1160.320,331.167,-76.108,-176.574,8.600,148.709
C03086=1160.316,331.414,-76.141,-176.572,8.603,148.709
C03087=1160.312,331.662,-76.173,-176.570,8.606,148.710
C03088=1160.308,331.910,-76.206,-176.568,8.610,148.710
C03089=1160.304,332.158,-76.239,-176.565,8.614,148.710
C03090=1160.299,332.406,-76.271,-176.562,8.617,148.710
C03091=1160.296,332.654,-76.304,-176.560,8.620,148.710
C03092=1160.291,332.901,-76.337,-176.557,8.623,148.710
C03093=1160.287,333.149,-76.369,-176.554,8.627,148.711
C03094=1160.283,333.397,-76.402,-176.552,8.631,148.711
C03095=1160.279,333.644,-76.435,-176.550,8.634,148.711
C03096=1160.275,333.892,-76.468,-176.547,8.638,148.711
C03097=1160.271,334.140,-76.500,-176.545,8.641,148.712
C03098=1160.267,334.388,-76.534,-176.542,8.645,148.712
C03099=1160.262,334.636,-76.567,-176.539,8.648,148.712
C03100=1160.258,334.883,-76.600,-176.537,8.652,148.712
C03101=1160.255,335.131,-76.632,-176.534,8.655,148.712
C03102=1160.251,335.379,-76.666,-176.532,8.658,148.712
C03103=1160.246,335.627,-76.698,-176.529,8.662,148.713
C03104=1160.242,335.875,-76.731,-176.527,8.666,148.713
C03105=1160.238,336.122,-76.764,-176.525,8.669,148.713
C03106=1160.234,336.370,-76.798,-176.522,8.673,148.713
C03107=1160.230,336.618,-76.831,-176.519,8.676,148.714
C03108=1160.226,336.866,-76.864,-176.517,8.680,148.714
C03109=1160.222,337.114,-76.897,-176.514,8.684,148.714
C03110=1160.218,337.362,-76.931,-176.512,8.687,148.714
C03111=1160.215,337.609,-76.963,-176.510,8.690,148.714
C03112=1160.210,337.857,-76.996,-176.507,8.694,148.715
C03113=1160.206,338.105,-77.029,-176.504,8.698,148.715
C03114=1160.202,338.352,-77.063,-176.502,8.701,148.715
C03115=1160.198,338.600,-77.096,-176.500,8.704,148.715
C03116=1160.194,338.848,-77.129,-176.497,8.708,148.715
C03117=1160.190,339.096,-77.162,-176.494,8.711,148.716
C03118=1160.185,339.375,-77.200,-176.491,8.715,148.716
C03119=1160.181,339.655,-77.237,-176.488,8.720,148.716
C03120=1160.176,339.935,-77.276,-176.486,8.724,148.716
C03121=1160.171,340.215,-77.313,-176.483,8.728,148.717
C03122=1160.167,340.463,-77.346,-176.480,8.731,148.717
C03123=1160.163,340.710,-77.379,-176.478,8.734,148.717
C03124=1160.159,340.958,-77.413,-176.475,8.738,148.717
C03125=1160.155,341.206,-77.446,-176.473,8.742,148.717
C03126=1160.151,341.454,-77.479,-176.471,8.745,148.718
C03127=1160.147,341.701,-77.513,-176.468,8.749,148.718
C03128=1160.143,341.948,-77.546,-176.465,8.752,148.718
C03129=1160.139,342.197,-77.579,-176.464,8.756,148.718
C03130=1160.134,342.445,-77.613,-176.461,8.760,148.719
C03131=1160.130,342.692,-77.647,-176.458,8.763,148.719
C03132=1160.126,342.940,-77.680,-176.456,8.767,148.719
C03133=1160.122,343.187,-77.713,-176.453,8.771,148.719
C03134=1160.118,343.435,-77.747,-176.451,8.774,148.720
C03135=1160.115,343.683,-77.781,-176.448,8.778,148.720
C03136=1160.111,343.931,-77.814,-176.446,8.781,148.720
C03137=1160.106,344.178,-77.848,-176.443,8.785,148.720
C03138=1160.102,344.426,-77.882,-176.440,8.789,148.721
C03139=1160.098,344.674,-77.915,-176.438,8.792,148.721
C03140=1160.094,344.921,-77.949,-176.436,8.795,148.721
C03141=1160.090,345.169,-77.982,-176.433,8.799,148.721
C03142=1160.085,345.417,-78.016,-176.431,8.803,148.721
C03143=1160.082,345.664,-78.050,-176.428,8.806,148.722
C03144=1160.077,345.912,-78.083,-176.426,8.810,148.722
C03145=1160.074,346.160,-78.117,-176.424,8.814,148.722
C03146=1160.069,346.408,-78.151,-176.421,8.818,148.723
C03147=1160.066,346.655,-78.185,-176.418,8.821,148.723
C03148=1160.061,346.903,-78.218,-176.416,8.824,148.723
C03149=1160.057,347.151,-78.253,-176.413,8.829,148.723
C03150=1160.053,347.399,-78.286,-176.411,8.832,148.723
C03151=1160.049,347.646,-78.320,-176.409,8.835,148.724
C03152=1160.045,347.893,-78.353,-176.406,8.839,148.724
C03153=1160.041,348.142,-78.388,-176.403,8.843,148.724
C03154=1160.037,348.389,-78.422,-176.401,8.847,148.725
C03155=1160.033,348.636,-78.455,-176.399,8.850,148.725
C03156=1160.029,348.884,-78.490,-176.396,8.854,148.725
C03157=1160.025,349.132,-78.523,-176.394,8.858,148.725
C03158=1160.021,349.380,-78.557,-176.391,8.861,148.725
C03159=1160.017,349.627,-78.591,-176.388,8.865,148.726
C03160=1160.013,349.875,-78.625,-176.386,8.868,148.726
C03161=1160.009,350.123,-78.659,-176.384,8.872,148.726
C03162=1160.005,350.370,-78.693,-176.381,8.876,148.727
C03163=1160.001,350.618,-78.728,-176.379,8.879,148.727
C03164=1159.997,350.866,-78.761,-176.376,8.883,148.727
C03165=1159.993,351.113,-78.795,-176.374,8.887,148.727
C03166=1159.989,351.361,-78.830,-176.371,8.891,148.728
C03167=1159.985,351.608,-78.864,-176.369,8.894,148.728
C03168=1159.981,351.857,-78.898,-176.367,8.898,148.728
C03169=1159.977,352.104,-78.931,-176.364,8.902,148.728
C03170=1159.972,352.351,-78.966,-176.362,8.905,148.729
C03171=1159.969,352.599,-79.000,-176.359,8.909,148.729
C03172=1159.965,352.846,-79.035,-176.357,8.913,148.729
C03173=1159.961,353.093,-79.069,-176.355,8.916,148.730
C03174=1159.957,353.342,-79.103,-176.352,8.920,148.730
C03175=1159.953,353.589,-79.137,-176.349,8.923,148.730
C03176=1159.949,353.837,-79.171,-176.347,8.928,148.731
C03177=1159.945,354.085,-79.205,-176.345,8.931,148.731
C03178=1159.940,354.332,-79.240,-176.342,8.935,148.731
C03179=1159.937,354.580,-79.274,-176.339,8.939,148.731
C03180=1159.933,354.827,-79.308,-176.337,8.943,148.732
C03181=1159.929,355.075,-79.343,-176.335,8.946,148.732
C03182=1159.925,355.322,-79.377,-176.332,8.949,148.732
C03183=1159.922,355.570,-79.411,-176.329,8.954,148.732
C03184=1159.917,355.818,-79.446,-176.328,8.957,148.733
C03185=1159.913,356.066,-79.481,-176.325,8.961,148.733
C03186=1159.909,356.313,-79.515,-176.322,8.965,148.733
C03187=1159.905,356.560,-79.549,-176.320,8.969,148.734
C03188=1159.901,356.808,-79.584,-176.318,8.972,148.734
C03189=1159.897,357.056,-79.618,-176.315,8.976,148.734
C03190=1159.893,357.304,-79.653,-176.312,8.980,148.734
C03191=1159.889,357.550,-79.687,-176.310,8.984,148.735
C03192=1159.885,357.798,-79.722,-176.308,8.987,148.735
C03193=1159.881,358.046,-79.756,-176.305,8.991,148.735
C03194=1159.878,358.294,-79.791,-176.303,8.995,148.736
C03195=1159.873,358.541,-79.825,-176.300,8.999,148.736
C03196=1159.869,358.789,-79.860,-176.298,9.002,148.736
C03197=1159.865,359.036,-79.895,-176.295,9.007,148.737
C03198=1159.862,359.284,-79.929,-176.293,9.010,148.737
C03199=1159.857,359.531,-79.964,-176.290,9.014,148.737
C03200=1159.853,359.779,-79.999,-176.288,9.018,148.738
C03201=1159.850,360.026,-80.034,-176.285,9.022,148.738
C03202=1159.845,360.274,-80.068,-176.283,9.025,148.738
C03203=1159.842,360.522,-80.103,-176.281,9.030,148.739
C03204=1159.837,360.769,-80.138,-176.278,9.033,148.739
C03205=1159.834,361.017,-80.172,-176.275,9.037,148.739
C03206=1159.829,361.264,-80.207,-176.274,9.041,148.740
C03207=1159.826,361.511,-80.242,-176.271,9.045,148.740
C03208=1159.822,361.760,-80.277,-176.268,9.048,148.740
C03209=1159.817,362.007,-80.312,-176.266,9.052,148.740
C03210=1159.814,362.254,-80.347,-176.264,9.056,148.741
C03211=1159.810,362.502,-80.381,-176.261,9.060,148.741
C03212=1159.806,362.749,-80.417,-176.258,9.064,148.741
C03213=1159.802,362.997,-80.451,-176.256,9.068,148.742
C03214=1159.798,363.245,-80.486,-176.253,9.072,148.742
C03215=1159.795,363.492,-80.521,-176.252,9.076,148.743
C03216=1159.790,363.739,-80.555,-176.249,9.080,148.743
C03217=1159.786,363.987,-80.591,-176.247,9.083,148.743
C03218=1159.782,364.235,-80.626,-176.244,9.087,148.744
C03219=1159.778,364.482,-80.661,-176.242,9.091,148.744
C03220=1159.774,364.729,-80.696,-176.239,9.095,148.744
C03221=1159.771,364.977,-80.731,-176.237,9.099,148.745
C03222=1159.766,365.260,-80.771,-176.234,9.104,148.745
C03223=1159.761,365.542,-80.811,-176.231,9.108,148.745
C03224=1159.757,365.825,-80.851,-176.229,9.112,148.746
C03225=1159.753,366.108,-80.892,-176.226,9.117,148.746
C03226=1159.749,366.355,-80.926,-176.224,9.121,148.747
C03227=1159.745,366.603,-80.962,-176.222,9.125,148.747
C03228=1159.741,366.850,-80.997,-176.219,9.129,148.747
C03229=1159.737,367.098,-81.032,-176.217,9.132,148.748
C03230=1159.733,367.345,-81.067,-176.215,9.137,148.748
C03231=1159.729,367.593,-81.103,-176.213,9.140,148.749
C03232=1159.725,367.839,-81.138,-176.210,9.144,148.749
C03233=1159.721,368.087,-81.173,-176.208,9.148,148.749
C03234=1159.718,368.335,-81.208,-176.206,9.152,148.750
C03235=1159.713,368.582,-81.244,-176.204,9.156,148.750
C03236=1159.709,368.830,-81.280,-176.202,9.160,148.751
C03237=1159.705,369.078,-81.314,-176.199,9.164,148.751
C03238=1159.701,369.325,-81.350,-176.197,9.168,148.752
C03239=1159.697,369.572,-81.385,-176.195,9.172,148.752
C03240=1159.693,369.820,-81.421,-176.193,9.176,148.752
C03241=1159.690,370.067,-81.456,-176.191,9.180,148.753
C03242=1159.686,370.315,-81.492,-176.189,9.184,148.753
C03243=1159.682,370.561,-81.527,-176.187,9.187,148.754
C03244=1159.678,370.809,-81.562,-176.184,9.192,148.754
C03245=1159.674,371.057,-81.597,-176.183,9.195,148.755
C03246=1159.670,371.305,-81.633,-176.181,9.199,148.755
C03247=1159.666,371.552,-81.669,-176.178,9.203,148.756
C03248=1159.662,371.799,-81.704,-176.176,9.207,148.756
C03249=1159.658,372.047,-81.740,-176.174,9.211,148.757
C03250=1159.654,372.294,-81.775,-176.172,9.215,148.757
C03251=1159.651,372.542,-81.811,-176.171,9.219,148.758
C03252=1159.646,372.789,-81.847,-176.169,9.222,148.758
C03253=1159.642,373.036,-81.882,-176.167,9.227,148.759
C03254=1159.639,373.284,-81.918,-176.165,9.231,148.759
C03255=1159.635,373.531,-81.953,-176.163,9.234,148.760
C03256=1159.631,373.779,-81.989,-176.161,9.238,148.760
C03257=1159.627,374.026,-82.025,-176.159,9.242,148.761
C03258=1159.623,374.274,-82.060,-176.158,9.246,148.761
C03259=1159.619,374.521,-82.096,-176.156,9.250,148.762
C03260=1159.615,374.768,-82.131,-176.154,9.254,148.762
C03261=1159.611,375.015,-82.168,-176.153,9.258,148.763
C03262=1159.607,375.263,-82.204,-176.150,9.262,148.763
C03263=1159.604,375.510,-82.239,-176.149,9.266,148.764
C03264=1159.600,375.758,-82.275,-176.147,9.270,148.765
C03265=1159.596,376.006,-82.311,-176.146,9.274,148.765
C03266=1159.591,376.253,-82.346,-176.144,9.277,148.766
C03267=1159.588,376.499,-82.382,-176.143,9.281,148.766
C03268=1159.584,376.747,-82.418,-176.141,9.285,148.767
C03269=1159.580,376.995,-82.454,-176.140,9.289,148.768
C03270=1159.576,377.242,-82.490,-176.138,9.293,148.768
C03271=1159.572,377.490,-82.526,-176.137,9.297,148.769
C03272=1159.569,377.737,-82.562,-176.135,9.301,148.769
C03273=1159.565,377.984,-82.597,-176.134,9.305,148.770
C03274=1159.561,378.232,-82.634,-176.133,9.309,148.771
C03275=1159.556,378.479,-82.669,-176.131,9.313,148.771
C03276=1159.553,378.726,-82.705,-176.130,9.316,148.772
C03277=1159.549,378.974,-82.741,-176.129,9.320,148.772
C03278=1159.545,379.221,-82.777,-176.128,9.324,148.773
C03279=1159.541,379.468,-82.813,-176.126,9.328,148.774
C03280=1159.537,379.716,-82.849,-176.125,9.332,148.775
C03281=1159.533,379.963,-82.885,-176.124,9.335,148.775
C03282=1159.529,380.211,-82.922,-176.123,9.339,148.776
C03283=1159.526,380.458,-82.957,-176.121,9.343,148.777
C03284=1159.522,380.706,-82.993,-176.121,9.346,148.777
C03285=1159.518,380.953,-83.030,-176.120,9.350,148.778
C03286=1159.514,381.200,-83.065,-176.119,9.354,148.779
C03287=1159.510,381.448,-83.102,-176.118,9.357,148.779
C03288=1159.506,381.695,-83.137,-176.117,9.362,148.780
C03289=1159.502,381.943,-83.174,-176.116,9.365,148.781
C03290=1159.499,382.190,-83.210,-176.115,9.369,148.782
C03291=1159.494,382.438,-83.246,-176.114,9.372,148.782
C03292=1159.491,382.684,-83.282,-176.113,9.375,148.783
C03293=1159.487,382.932,-83.318,-176.112,9.379,148.784
C03294=1159.483,383.178,-83.354,-176.112,9.383,148.784
C03295=1159.479,383.426,-83.390,-176.112,9.386,148.785
C03296=1159.475,383.673,-83.427,-176.111,9.390,148.786
C03297=1159.471,383.921,-83.462,-176.110,9.394,148.787
C03298=1159.467,384.168,-83.499,-176.110,9.397,148.788
C03299=1159.463,384.415,-83.535,-176.109,9.400,148.788
C03300=1159.459,384.662,-83.572,-176.108,9.404,148.789
C03301=1159.456,384.910,-83.607,-176.108,9.407,148.790
C03302=1159.452,385.157,-83.644,-176.108,9.411,148.791
C03303=1159.448,385.405,-83.679,-176.107,9.414,148.791
C03304=1159.444,385.652,-83.716,-176.107,9.418,148.792
C03305=1159.440,385.899,-83.752,-176.107,9.421,148.793
C03306=1159.436,386.147,-83.789,-176.106,9.424,148.794
C03307=1159.433,386.394,-83.826,-176.106,9.428,148.794
C03308=1159.429,386.642,-83.862,-176.106,9.431,148.795
C03309=1159.425,386.889,-83.898,-176.106,9.434,148.796
C03310=1159.421,387.137,-83.934,-176.105,9.437,148.797
C03311=1159.417,387.384,-83.971,-176.105,9.441,148.798
C03312=1159.413,387.631,-84.006,-176.105,9.444,148.799
C03313=1159.409,387.879,-84.043,-176.105,9.447,148.799
C03314=1159.406,388.125,-84.079,-176.105,9.450,148.800
C03315=1159.402,388.373,-84.116,-176.105,9.453,148.801
C03316=1159.398,388.620,-84.152,-176.105,9.456,148.802
C03317=1159.394,388.867,-84.189,-176.105,9.460,148.803
C03318=1159.390,389.115,-84.225,-176.105,9.462,148.803
C03319=1159.386,389.362,-84.261,-176.106,9.465,148.804
C03320=1159.382,389.609,-84.298,-176.105,9.468,148.805
C03321=1159.379,389.857,-84.334,-176.106,9.471,148.806
C03322=1159.375,390.104,-84.370,-176.106,9.474,148.807
C03323=1159.371,390.351,-84.407,-176.106,9.476,148.807
C03324=1159.367,390.599,-84.443,-176.107,9.479,148.808
C03325=1159.363,390.846,-84.480,-176.107,9.483,148.809
C03326=1159.358,391.131,-84.521,-176.107,9.486,148.810
C03327=1159.354,391.418,-84.564,-176.108,9.489,148.811
C03328=1159.350,391.703,-84.606,-176.108,9.492,148.812
C03329=1159.345,391.989,-84.648,-176.108,9.495,148.813
C03330=1159.342,392.236,-84.684,-176.108,9.498,148.814
C03331=1159.338,392.483,-84.721,-176.109,9.501,148.815
C03332=1159.333,392.731,-84.757,-176.110,9.504,148.815
C03333=1159.330,392.978,-84.793,-176.110,9.506,148.816
C03334=1159.326,393.225,-84.830,-176.110,9.509,148.817
C03335=1159.322,393.472,-84.866,-176.111,9.511,148.818
C03336=1159.318,393.719,-84.903,-176.112,9.514,148.819
C03337=1159.314,393.967,-84.939,-176.112,9.516,148.819
C03338=1159.311,394.214,-84.975,-176.112,9.519,148.820
C03339=1159.307,394.462,-85.013,-176.113,9.521,148.821
C03340=1159.303,394.710,-85.049,-176.113,9.524,148.822
C03341=1159.299,394.957,-85.085,-176.114,9.527,148.823
C03342=1159.295,395.204,-85.122,-176.115,9.528,148.823
C03343=1159.292,395.451,-85.158,-176.115,9.531,148.824
C03344=1159.287,395.699,-85.194,-176.115,9.534,148.825
C03345=1159.283,395.946,-85.231,-176.117,9.536,148.826
C03346=1159.280,396.193,-85.267,-176.117,9.538,148.826
C03347=1159.276,396.440,-85.304,-176.118,9.540,148.827
C03348=1159.271,396.688,-85.340,-176.118,9.543,148.828
C03349=1159.268,396.935,-85.377,-176.118,9.546,148.829
C03350=1159.264,397.182,-85.414,-176.120,9.548,148.830
C03351=1159.260,397.429,-85.450,-176.120,9.550,148.830
C03352=1159.256,397.676,-85.486,-176.121,9.553,148.831
C03353=1159.253,397.924,-85.523,-176.122,9.554,148.832
C03354=1159.249,398.171,-85.560,-176.122,9.557,148.833
C03355=1159.245,398.418,-85.596,-176.123,9.559,148.834
C03356=1159.241,398.666,-85.632,-176.123,9.561,148.834
C03357=1159.237,398.913,-85.669,-176.124,9.564,148.835
C03358=1159.233,399.160,-85.706,-176.125,9.565,148.836
C03359=1159.229,399.407,-85.742,-176.125,9.568,148.837
C03360=1159.225,399.655,-85.779,-176.126,9.570,148.837
C03361=1159.222,399.902,-85.815,-176.127,9.572,148.838
C03362=1159.218,400.149,-85.852,-176.127,9.575,148.839
C03363=1159.213,400.397,-85.889,-176.128,9.577,148.840
C03364=1159.210,400.643,-85.925,-176.129,9.578,148.840
C03365=1159.206,400.892,-85.961,-176.129,9.581,148.841
C03366=1159.202,401.139,-85.998,-176.130,9.583,148.842
C03367=1159.199,401.386,-86.034,-176.131,9.585,148.843
C03368=1159.195,401.633,-86.071,-176.132,9.586,148.843
C03369=1159.190,401.881,-86.107,-176.132,9.589,148.844
C03370=1159.187,402.128,-86.144,-176.133,9.591,148.845
C03371=1159.183,402.375,-86.181,-176.134,9.593,148.845
C03372=1159.179,402.622,-86.217,-176.135,9.595,148.846
C03373=1159.175,402.869,-86.254,-176.135,9.597,148.847
C03374=1159.171,403.117,-86.290,-176.136,9.599,148.848
C03375=1159.168,403.365,-86.327,-176.136,9.601,148.848
C03376=1159.164,403.612,-86.363,-176.137,9.603,148.849
C03377=1159.160,403.859,-86.400,-176.138,9.605,148.850
C03378=1159.156,404.106,-86.437,-176.139,9.607,148.850
C03379=1159.152,404.354,-86.473,-176.140,9.608,148.851
C03380=1159.148,404.601,-86.509,-176.140,9.611,148.852
C03381=1159.144,404.848,-86.546,-176.141,9.613,148.853
C03382=1159.141,405.095,-86.583,-176.141,9.615,148.853
C03383=1159.137,405.342,-86.619,-176.142,9.616,148.854
C03384=1159.132,405.590,-86.656,-176.143,9.618,148.854
C03385=1159.130,405.837,-86.692,-176.144,9.620,148.855
C03386=1159.125,406.085,-86.729,-176.145,9.622,148.856
C03387=1159.121,406.332,-86.766,-176.145,9.625,148.857
C03388=1159.118,406.579,-86.802,-176.145,9.626,148.857
C03389=1159.114,406.826,-86.838,-176.146,9.628,148.858
C03390=1159.109,407.074,-86.875,-176.147,9.630,148.859
C03391=1159.105,407.321,-86.912,-176.148,9.632,148.859
C03392=1159.102,407.568,-86.948,-176.148,9.633,148.860
C03393=1159.098,407.815,-86.985,-176.149,9.635,148.861
C03394=1159.094,408.062,-87.022,-176.150,9.637,148.861
C03395=1159.091,408.310,-87.058,-176.150,9.638,148.862
C03396=1159.087,408.558,-87.095,-176.151,9.640,148.862
C03397=1159.083,408.805,-87.132,-176.151,9.643,148.863
C03398=1159.079,409.052,-87.168,-176.152,9.645,148.864
C03399=1159.075,409.299,-87.205,-176.153,9.646,148.864
C03400=1159.071,409.546,-87.242,-176.153,9.648,148.865
C03401=1159.067,409.793,-87.277,-176.154,9.650,148.866
C03402=1159.063,410.041,-87.314,-176.155,9.652,148.866
C03403=1159.059,410.288,-87.351,-176.155,9.653,148.867
C03404=1159.056,410.536,-87.388,-176.156,9.655,148.868
C03405=1159.052,410.783,-87.424,-176.157,9.657,148.868
C03406=1159.048,411.030,-87.461,-176.157,9.659,148.869
C03407=1159.044,411.278,-87.497,-176.158,9.661,148.870
C03408=1159.040,411.525,-87.534,-176.158,9.663,148.870
C03409=1159.036,411.772,-87.571,-176.158,9.664,148.871
C03410=1159.032,412.019,-87.607,-176.159,9.666,148.871
C03411=1159.028,412.266,-87.644,-176.160,9.668,148.872
C03412=1159.025,412.513,-87.680,-176.161,9.670,148.873
C03413=1159.021,412.761,-87.717,-176.161,9.671,148.873
C03414=1159.017,413.009,-87.754,-176.162,9.673,148.874
C03415=1159.014,413.256,-87.790,-176.162,9.674,148.874
C03416=1159.009,413.503,-87.827,-176.162,9.677,148.875
C03417=1159.005,413.750,-87.864,-176.163,9.679,148.876
C03418=1159.001,413.997,-87.901,-176.164,9.681,148.876
C03419=1158.998,414.244,-87.937,-176.164,9.682,148.877
C03420=1158.994,414.492,-87.973,-176.165,9.684,148.878
C03421=1158.989,414.739,-88.010,-176.165,9.685,148.878
C03422=1158.987,414.987,-88.047,-176.166,9.687,148.879
C03423=1158.983,415.234,-88.083,-176.166,9.689,148.879
C03424=1158.981,415.481,-88.119,-176.166,9.691,148.880
C03425=1158.979,415.728,-88.156,-176.167,9.693,148.881
C03426=1158.978,416.101,-88.211,-176.168,9.695,148.881
C03427=1158.978,416.473,-88.265,-176.168,9.698,148.882
C03428=1158.982,416.846,-88.319,-176.169,9.700,148.883
C03429=1158.986,417.217,-88.373,-176.170,9.703,148.884
C03430=1158.565,417.219,-88.420,-176.172,9.714,148.888
C03431=1158.560,416.844,-88.366,-176.172,9.711,148.887
C03432=1158.558,416.468,-88.312,-176.171,9.709,148.886
C03433=1158.557,416.093,-88.257,-176.170,9.707,148.885
C03434=1158.557,415.716,-88.202,-176.170,9.704,148.884
C03435=1158.559,415.470,-88.165,-176.169,9.702,148.884
C03436=1158.562,415.222,-88.128,-176.169,9.700,148.883
C03437=1158.565,414.975,-88.092,-176.168,9.699,148.882
C03438=1158.569,414.728,-88.055,-176.168,9.696,148.882
C03439=1158.573,414.481,-88.018,-176.167,9.694,148.881
C03440=1158.577,414.233,-87.981,-176.167,9.693,148.881
C03441=1158.581,413.985,-87.946,-176.166,9.691,148.880
C03442=1158.585,413.738,-87.909,-176.166,9.689,148.879
C03443=1158.589,413.491,-87.872,-176.165,9.688,148.879
C03444=1158.592,413.244,-87.836,-176.164,9.686,148.878
C03445=1158.596,412.997,-87.799,-176.165,9.684,148.878
C03446=1158.600,412.750,-87.762,-176.164,9.682,148.877
C03447=1158.604,412.503,-87.725,-176.163,9.680,148.876
C03448=1158.608,412.255,-87.689,-176.163,9.678,148.876
C03449=1158.612,412.007,-87.652,-176.162,9.677,148.875
C03450=1158.616,411.760,-87.615,-176.161,9.675,148.874
C03451=1158.619,411.513,-87.579,-176.161,9.674,148.874
C03452=1158.623,411.266,-87.542,-176.160,9.672,148.873
C03453=1158.627,411.019,-87.505,-176.160,9.670,148.873
C03454=1158.631,410.772,-87.469,-176.159,9.668,148.872
C03455=1158.635,410.524,-87.433,-176.159,9.666,148.871
C03456=1158.639,410.277,-87.396,-176.158,9.664,148.871
C03457=1158.643,410.030,-87.359,-176.157,9.662,148.870
C03458=1158.646,409.782,-87.323,-176.157,9.660,148.869
C03459=1158.650,409.535,-87.286,-176.156,9.659,148.869
C03460=1158.654,409.288,-87.249,-176.155,9.657,148.868
C03461=1158.658,409.040,-87.213,-176.155,9.655,148.867
C03462=1158.662,408.793,-87.176,-176.154,9.653,148.867
C03463=1158.666,408.546,-87.140,-176.153,9.652,148.866
C03464=1158.670,408.299,-87.103,-176.153,9.650,148.865
C03465=1158.673,408.052,-87.067,-176.152,9.648,148.865
C03466=1158.677,407.804,-87.029,-176.152,9.646,148.864
C03467=1158.681,407.556,-86.993,-176.151,9.644,148.863
C03468=1158.685,407.309,-86.957,-176.150,9.642,148.863
C03469=1158.689,407.062,-86.920,-176.150,9.640,148.862
C03470=1158.693,406.815,-86.883,-176.149,9.639,148.861
C03471=1158.696,406.568,-86.847,-176.148,9.637,148.861
C03472=1158.700,406.321,-86.810,-176.147,9.635,148.860
C03473=1158.705,406.073,-86.774,-176.146,9.633,148.859
C03474=1158.709,405.826,-86.737,-176.146,9.631,148.859
C03475=1158.712,405.579,-86.701,-176.145,9.630,148.858
C03476=1158.716,405.331,-86.664,-176.145,9.627,148.857
C03477=1158.720,405.084,-86.627,-176.144,9.625,148.857
C03478=1158.723,404.837,-86.590,-176.143,9.623,148.856
C03479=1158.727,404.589,-86.554,-176.142,9.622,148.855
C03480=1158.732,404.342,-86.517,-176.142,9.620,148.855
C03481=1158.735,404.095,-86.481,-176.141,9.618,148.854
C03482=1158.739,403.848,-86.444,-176.140,9.616,148.853
C03483=1158.743,403.601,-86.407,-176.140,9.613,148.852
C03484=1158.747,403.353,-86.372,-176.139,9.612,148.852
C03485=1158.750,403.105,-86.335,-176.138,9.610,148.851
C03486=1158.754,402.858,-86.298,-176.137,9.608,148.850
C03487=1158.758,402.611,-86.262,-176.137,9.606,148.850
C03488=1158.762,402.364,-86.225,-176.136,9.604,148.849
C03489=1158.766,402.116,-86.189,-176.136,9.602,148.848
C03490=1158.770,401.869,-86.152,-176.135,9.600,148.847
C03491=1158.774,401.622,-86.115,-176.134,9.598,148.847
C03492=1158.778,401.375,-86.079,-176.133,9.596,148.846
C03493=1158.782,401.128,-86.042,-176.133,9.593,148.845
C03494=1158.785,400.880,-86.006,-176.132,9.592,148.845
C03495=1158.790,400.633,-85.969,-176.131,9.590,148.844
C03496=1158.793,400.385,-85.932,-176.130,9.588,148.843
C03497=1158.796,400.138,-85.896,-176.130,9.585,148.842
C03498=1158.801,399.891,-85.859,-176.129,9.583,148.842
C03499=1158.805,399.643,-85.823,-176.128,9.581,148.841
C03500=1158.808,399.396,-85.787,-176.128,9.579,148.840
C03501=1158.812,399.149,-85.750,-176.127,9.577,148.839
C03502=1158.816,398.902,-85.713,-176.126,9.575,148.838
C03503=1158.820,398.655,-85.677,-176.126,9.572,148.838
C03504=1158.824,398.407,-85.640,-176.125,9.570,148.837
C03505=1158.828,398.160,-85.604,-176.124,9.568,148.836
C03506=1158.832,397.913,-85.567,-176.123,9.565,148.835
C03507=1158.835,397.665,-85.530,-176.123,9.564,148.835
C03508=1158.840,397.417,-85.494,-176.122,9.561,148.834
C03509=1158.843,397.171,-85.458,-176.121,9.559,148.833
C03510=1158.847,396.923,-85.421,-176.121,9.556,148.832
C03511=1158.851,396.676,-85.384,-176.120,9.554,148.832
C03512=1158.855,396.429,-85.348,-176.120,9.552,148.831
C03513=1158.859,396.182,-85.312,-176.118,9.550,148.830
C03514=1158.862,395.935,-85.275,-176.118,9.547,148.829
C03515=1158.866,395.687,-85.238,-176.117,9.545,148.828
C03516=1158.871,395.440,-85.202,-176.117,9.542,148.828
C03517=1158.874,395.193,-85.166,-176.117,9.540,148.827
C03518=1158.878,394.946,-85.129,-176.116,9.538,148.826
C03519=1158.882,394.698,-85.092,-176.115,9.535,148.825
C03520=1158.885,394.450,-85.056,-176.115,9.532,148.824
C03521=1158.889,394.203,-85.020,-176.114,9.530,148.824
C03522=1158.894,393.956,-84.983,-176.113,9.527,148.823
C03523=1158.897,393.709,-84.946,-176.113,9.525,148.822
C03524=1158.901,393.461,-84.910,-176.113,9.522,148.821
C03525=1158.905,393.214,-84.873,-176.112,9.520,148.820
C03526=1158.909,392.967,-84.837,-176.112,9.517,148.820
C03527=1158.913,392.720,-84.800,-176.111,9.514,148.819
C03528=1158.916,392.472,-84.765,-176.111,9.512,148.818
C03529=1158.921,392.225,-84.728,-176.110,9.509,148.817
C03530=1158.925,391.978,-84.691,-176.110,9.506,148.816
C03531=1158.928,391.692,-84.649,-176.109,9.503,148.815
C03532=1158.933,391.406,-84.607,-176.109,9.500,148.814
C03533=1158.937,391.120,-84.565,-176.109,9.497,148.813
C03534=1158.942,390.834,-84.523,-176.108,9.494,148.812
C03535=1158.946,390.587,-84.487,-176.108,9.491,148.812
C03536=1158.950,390.340,-84.450,-176.108,9.488,148.811
C03537=1158.954,390.092,-84.414,-176.108,9.485,148.810
C03538=1158.958,389.846,-84.378,-176.107,9.482,148.809
C03539=1158.962,389.598,-84.341,-176.107,9.480,148.808
C03540=1158.965,389.351,-84.305,-176.107,9.477,148.808
C03541=1158.969,389.104,-84.268,-176.107,9.473,148.807
C03542=1158.973,388.856,-84.231,-176.107,9.470,148.806
C03543=1158.977,388.608,-84.196,-176.107,9.467,148.805
C03544=1158.981,388.361,-84.159,-176.106,9.464,148.804
C03545=1158.984,388.114,-84.123,-176.106,9.462,148.804
C03546=1158.988,387.866,-84.086,-176.106,9.458,148.803
C03547=1158.992,387.619,-84.050,-176.107,9.455,148.802
C03548=1158.996,387.372,-84.013,-176.107,9.452,148.801
C03549=1159.000,387.124,-83.977,-176.107,9.448,148.800
C03550=1159.004,386.878,-83.941,-176.107,9.446,148.799
C03551=1159.008,386.630,-83.905,-176.107,9.442,148.799
C03552=1159.011,386.383,-83.868,-176.107,9.439,148.798
C03553=1159.015,386.136,-83.832,-176.107,9.435,148.797
C03554=1159.019,385.888,-83.796,-176.108,9.432,148.796
C03555=1159.023,385.641,-83.759,-176.108,9.429,148.795
C03556=1159.027,385.394,-83.724,-176.108,9.426,148.795
C03557=1159.031,385.146,-83.687,-176.109,9.422,148.794
C03558=1159.035,384.899,-83.651,-176.109,9.419,148.793
C03559=1159.039,384.652,-83.614,-176.110,9.416,148.792
C03560=1159.042,384.405,-83.578,-176.111,9.412,148.792
C03561=1159.046,384.157,-83.542,-176.111,9.408,148.791
C03562=1159.050,383.910,-83.506,-176.111,9.405,148.790
C03563=1159.054,383.662,-83.470,-176.112,9.401,148.789
C03564=1159.058,383.415,-83.433,-176.112,9.398,148.789
C03565=1159.062,383.168,-83.397,-176.113,9.394,148.788
C03566=1159.065,382.921,-83.361,-176.114,9.390,148.787
C03567=1159.070,382.673,-83.325,-176.115,9.387,148.786
C03568=1159.073,382.426,-83.288,-176.116,9.383,148.786
C03569=1159.078,382.178,-83.252,-176.116,9.380,148.785
C03570=1159.081,381.931,-83.217,-176.118,9.376,148.784
C03571=1159.085,381.684,-83.180,-176.118,9.372,148.783
C03572=1159.089,381.436,-83.144,-176.119,9.368,148.783
C03573=1159.093,381.189,-83.108,-176.120,9.365,148.782
C03574=1159.097,380.941,-83.072,-176.121,9.361,148.781
C03575=1159.100,380.694,-83.036,-176.122,9.358,148.781
C03576=1159.104,380.447,-83.000,-176.123,9.354,148.780
C03577=1159.108,380.199,-82.964,-176.124,9.350,148.779
C03578=1159.112,379.952,-82.927,-176.125,9.347,148.779
C03579=1159.116,379.704,-82.892,-176.126,9.342,148.778
C03580=1159.121,379.457,-82.856,-176.128,9.339,148.777
C03581=1159.124,379.210,-82.820,-176.129,9.335,148.777
C03582=1159.128,378.963,-82.784,-176.131,9.331,148.776
C03583=1159.132,378.715,-82.748,-176.131,9.327,148.775
C03584=1159.136,378.468,-82.712,-176.132,9.323,148.775
C03585=1159.139,378.221,-82.676,-176.134,9.320,148.774
C03586=1159.144,377.973,-82.640,-176.135,9.316,148.773
C03587=1159.147,377.726,-82.604,-176.137,9.312,148.773
C03588=1159.151,377.478,-82.568,-176.138,9.308,148.772
C03589=1159.155,377.231,-82.532,-176.140,9.304,148.771
C03590=1159.159,376.983,-82.496,-176.141,9.300,148.771
C03591=1159.164,376.736,-82.461,-176.143,9.296,148.770
C03592=1159.167,376.489,-82.424,-176.144,9.292,148.770
C03593=1159.171,376.242,-82.389,-176.146,9.289,148.769
C03594=1159.174,375.994,-82.353,-176.147,9.285,148.768
C03595=1159.179,375.746,-82.317,-176.149,9.281,148.768
C03596=1159.183,375.499,-82.282,-176.150,9.277,148.767
C03597=1159.186,375.252,-82.245,-176.153,9.273,148.767
C03598=1159.190,375.004,-82.209,-176.154,9.269,148.766
C03599=1159.195,374.757,-82.174,-176.156,9.265,148.766
C03600=1159.198,374.510,-82.138,-176.158,9.261,148.765
C03601=1159.202,374.262,-82.103,-176.159,9.257,148.764
C03602=1159.206,374.015,-82.067,-176.161,9.253,148.764
C03603=1159.210,373.767,-82.031,-176.163,9.249,148.763
C03604=1159.214,373.520,-81.996,-176.165,9.245,148.763
C03605=1159.217,373.272,-81.960,-176.167,9.242,148.763
C03606=1159.222,373.025,-81.925,-176.169,9.237,148.762
C03607=1159.226,372.778,-81.889,-176.171,9.233,148.761
C03608=1159.230,372.530,-81.853,-176.172,9.230,148.761
C03609=1159.233,372.283,-81.818,-176.174,9.226,148.760
C03610=1159.237,372.035,-81.782,-176.176,9.222,148.760
C03611=1159.241,371.788,-81.747,-176.178,9.218,148.759
C03612=1159.246,371.540,-81.711,-176.181,9.214,148.759
C03613=1159.249,371.293,-81.675,-176.183,9.210,148.759
C03614=1159.253,371.045,-81.640,-176.184,9.206,148.758
C03615=1159.257,370.798,-81.604,-176.186,9.202,148.757
C03616=1159.261,370.551,-81.569,-176.188,9.198,148.757
C03617=1159.264,370.304,-81.533,-176.191,9.194,148.757
C03618=1159.268,370.056,-81.498,-176.193,9.190,148.756
C03619=1159.272,369.809,-81.462,-176.195,9.186,148.756
C03620=1159.276,369.562,-81.427,-176.197,9.182,148.755
C03621=1159.281,369.313,-81.392,-176.199,9.178,148.755
C03622=1159.284,369.066,-81.356,-176.201,9.174,148.754
C03623=1159.288,368.818,-81.321,-176.204,9.171,148.754
C03624=1159.292,368.572,-81.285,-176.206,9.166,148.754
C03625=1159.296,368.324,-81.250,-176.208,9.163,148.753
C03626=1159.300,368.076,-81.215,-176.210,9.158,148.753
C03627=1159.304,367.828,-81.180,-176.212,9.155,148.752
C03628=1159.308,367.582,-81.144,-176.215,9.150,148.752
C03629=1159.312,367.334,-81.109,-176.217,9.147,148.752
C03630=1159.316,367.086,-81.074,-176.219,9.143,148.751
C03631=1159.320,366.839,-81.039,-176.221,9.139,148.751
C03632=1159.323,366.592,-81.003,-176.224,9.135,148.750
C03633=1159.327,366.344,-80.968,-176.226,9.131,148.750
C03634=1159.332,366.097,-80.933,-176.229,9.127,148.750
C03635=1159.335,365.814,-80.893,-176.231,9.123,148.749
C03636=1159.340,365.531,-80.853,-176.234,9.118,148.749
C03637=1159.345,365.249,-80.813,-176.236,9.114,148.748
C03638=1159.350,364.966,-80.772,-176.239,9.110,148.748
C03639=1159.354,364.718,-80.738,-176.242,9.105,148.748
C03640=1159.357,364.470,-80.702,-176.244,9.102,148.747
C03641=1159.361,364.223,-80.668,-176.246,9.098,148.747
C03642=1159.365,363.976,-80.633,-176.249,9.093,148.746
C03643=1159.369,363.728,-80.598,-176.251,9.090,148.746
C03644=1159.373,363.481,-80.563,-176.254,9.086,148.746
C03645=1159.377,363.233,-80.528,-176.256,9.082,148.746
C03646=1159.381,362.985,-80.492,-176.259,9.078,148.745
C03647=1159.385,362.738,-80.458,-176.261,9.075,148.745
C03648=1159.388,362.491,-80.423,-176.264,9.071,148.745
C03649=1159.393,362.243,-80.388,-176.266,9.067,148.744
C03650=1159.396,361.996,-80.353,-176.268,9.063,148.744
C03651=1159.400,361.748,-80.318,-176.271,9.058,148.743
C03652=1159.405,361.500,-80.283,-176.273,9.055,148.743
C03653=1159.408,361.253,-80.249,-176.276,9.051,148.743
C03654=1159.412,361.006,-80.214,-176.278,9.047,148.743
C03655=1159.416,360.758,-80.179,-176.281,9.043,148.742
C03656=1159.421,360.511,-80.144,-176.283,9.040,148.742
C03657=1159.425,360.263,-80.109,-176.286,9.036,148.742
C03658=1159.428,360.015,-80.075,-176.288,9.032,148.741
C03659=1159.432,359.768,-80.040,-176.291,9.028,148.741
C03660=1159.436,359.520,-80.005,-176.293,9.025,148.741
C03661=1159.440,359.273,-79.971,-176.296,9.021,148.740
